TYPE "UDT_VfdNordParameter"
TITLE = UDT_VfdNordParameter
VERSION : 0.1
//Parameter structure to read and write
   STRUCT
      WriteValue : DInt;   // Parameter value to write
      ActualValue : DInt;   // Actual value read from VFD
      ParaNumber : Int;   // Parameter number to access
      Index : Int;   // Parameter index number to access
      ParaSet : Int;   // Parameter set to acces
      Format32 { ExternalAccessible := 'False'; ExternalVisible := 'False'; ExternalWritable := 'False'} : Bool;   // 1 = Write the parameter in DWord format. 0 = Write the parameter in Word format
      WriteAccess { ExternalAccessible := 'False'; ExternalVisible := 'False'; ExternalWritable := 'False'} : Bool;   // 1 = Write the parameter. 0 = Read the parameter
      InUse { ExternalAccessible := 'False'; ExternalVisible := 'False'; ExternalWritable := 'False'} : Bool;   // 1 = Parameter is to be processed
      RamOnly { ExternalAccessible := 'False'; ExternalVisible := 'False'; ExternalWritable := 'False'} : Bool;   // 1 = Save parameter in RAM, 0 = Save parameter in RAM and EEPROM
   END_STRUCT;

END_TYPE

FUNCTION_BLOCK "FB_VfdNORDParaAcycWrite"
{ S7_Optimized_Access := 'FALSE' }
VERSION : 0.1
// ATTRIBUTES
// AUTO_NUMBER = True
// BLOCK_NUMBER = 35
// END_ATTRIBUTES
   VAR_INPUT
      HW_Identifier { ExternalAccessible := 'False'; ExternalVisible := 'False'; ExternalWritable := 'False'} : HW_IO;
      idi_Value { ExternalAccessible := 'False'; ExternalVisible := 'False'; ExternalWritable := 'False'} : DInt;
      ii_FISystembus { ExternalAccessible := 'False'; ExternalVisible := 'False'; ExternalWritable := 'False'} : Int := 1;
      ii_ParameterNumber { ExternalAccessible := 'False'; ExternalVisible := 'False'; ExternalWritable := 'False'} : Int;
      ii_ParameterIndex { ExternalAccessible := 'False'; ExternalVisible := 'False'; ExternalWritable := 'False'} : Int;
      ii_ParameterSet { ExternalAccessible := 'False'; ExternalVisible := 'False'; ExternalWritable := 'False'} : Int;
      ix_Execute { ExternalAccessible := 'False'; ExternalVisible := 'False'; ExternalWritable := 'False'} : Bool;
      ix_Parameter32Bit { ExternalAccessible := 'False'; ExternalVisible := 'False'; ExternalWritable := 'False'} : Bool;
      ix_RAM_Only { ExternalAccessible := 'False'; ExternalVisible := 'False'; ExternalWritable := 'False'} : Bool;
   END_VAR

   VAR_OUTPUT
      qx_Done { ExternalAccessible := 'False'; ExternalVisible := 'False'; ExternalWritable := 'False'} : Bool;
      qx_Busy { ExternalAccessible := 'False'; ExternalVisible := 'False'; ExternalWritable := 'False'} : Bool;
      qx_Error { ExternalAccessible := 'False'; ExternalVisible := 'False'; ExternalWritable := 'False'} : Bool;
      qdi_ValueRead { ExternalAccessible := 'False'; ExternalVisible := 'False'; ExternalWritable := 'False'} : DInt;
      qw_ErrorID { ExternalAccessible := 'False'; ExternalVisible := 'False'; ExternalWritable := 'False'} : Word;
   END_VAR

   VAR
      sa_WriteVal { ExternalAccessible := 'False'; ExternalVisible := 'False'; ExternalWritable := 'False'} : Array[0..3] of Word;
      sa_RecWrite { ExternalAccessible := 'False'; ExternalVisible := 'False'; ExternalWritable := 'False'} AT sa_WriteVal : Struct
         PKE { ExternalAccessible := 'False'; ExternalVisible := 'False'; ExternalWritable := 'False'} : Word;
         Index { ExternalAccessible := 'False'; ExternalVisible := 'False'; ExternalWritable := 'False'} : Word;
         Para_Val { ExternalAccessible := 'False'; ExternalVisible := 'False'; ExternalWritable := 'False'} : DInt;
      END_STRUCT;
      sa_ReadVal { ExternalAccessible := 'False'; ExternalVisible := 'False'; ExternalWritable := 'False'} : Array[0..3] of Word;
      sa_RecRead { ExternalAccessible := 'False'; ExternalVisible := 'False'; ExternalWritable := 'False'} AT sa_ReadVal : Struct
         PKE { ExternalAccessible := 'False'; ExternalVisible := 'False'; ExternalWritable := 'False'} : Word;
         Index { ExternalAccessible := 'False'; ExternalVisible := 'False'; ExternalWritable := 'False'} : Word;
         Para_Val { ExternalAccessible := 'False'; ExternalVisible := 'False'; ExternalWritable := 'False'} : DInt;
      END_STRUCT;
      sv_WRRECInstance {InstructionName := 'WRREC'; LibVersion := '1.1'; ExternalAccessible := 'False'; ExternalVisible := 'False'; ExternalWritable := 'False'; S7_SetPoint := 'False'} : WRREC;
      sv_RDRECInstance {InstructionName := 'RDREC'; LibVersion := '1.0'; ExternalAccessible := 'False'; ExternalVisible := 'False'; ExternalWritable := 'False'; S7_SetPoint := 'False'} : RDREC;
      sw_Ak { ExternalAccessible := 'False'; ExternalVisible := 'False'; ExternalWritable := 'False'} : Word;
      sw_Pnu { ExternalAccessible := 'False'; ExternalVisible := 'False'; ExternalWritable := 'False'} : Word;
      sw_ErrorIDStatic { ExternalAccessible := 'False'; ExternalVisible := 'False'; ExternalWritable := 'False'} : Word;
      sdi_DataRecord { ExternalAccessible := 'False'; ExternalVisible := 'False'; ExternalWritable := 'False'} : DInt;
      si_Receivecounter { ExternalAccessible := 'False'; ExternalVisible := 'False'; ExternalWritable := 'False'} : Int;
      si_State { ExternalAccessible := 'False'; ExternalVisible := 'False'; ExternalWritable := 'False'} : Int;
      sx_FLMExecute { ExternalAccessible := 'False'; ExternalVisible := 'False'; ExternalWritable := 'False'} : Bool;
      sx_REdgeExecute { ExternalAccessible := 'False'; ExternalVisible := 'False'; ExternalWritable := 'False'} : Bool;
      sx_DoneStatic { ExternalAccessible := 'False'; ExternalVisible := 'False'; ExternalWritable := 'False'} : Bool;
      sx_ErrorStatic { ExternalAccessible := 'False'; ExternalVisible := 'False'; ExternalWritable := 'False'} : Bool;
   END_VAR

   VAR_TEMP
      tw_ResponseIND : Word;
      tw_ResponseLABEL : Word;
      tw_ResponsePNU : Word;
      tdi_ResponsePWE : DInt;
      tx_WithIndex : Bool;
      tx_WithParameterSet : Bool;
   END_VAR

   VAR CONSTANT
      cw_ChangeParameterValueWordEEPROM : Word := 2;
      cw_ChangeParameterValueWordRAM : Word := 14;
      cw_ChangeParameterValueDoubleWordEEPROM : Word := 3;
      cw_ChangeParameterValueDoubleWordRAM : Word := 13;
      cw_IncorretSubindex : Word := 3;
      cw_InternalResponseLabelCannotBeDepicted : Word := 202;
      cw_InvalidDataType : Word := 5;
      cw_NoResponse : Word := 0;
      cw_OrderCannotBeExecuted : Word := 7;
      cw_ParameterOffset : Word := 1000;
      cw_PNUMask : Word := 16#07FF;
      ci_ReceivecounterMax : Int := 255;
      ci_Length : UInt := 8;
   END_VAR


BEGIN
	(*
	----------------------------------------------------------------------------------------

	Version history:
	Date        | Version   | Author        | Remark
	----------------------------------------------------------------------------------------
	25/01/2021  | 0.1       | S.Theocharis  | Copy fron NORD library
	21/02/2023  | 4.0       | F.Baten       | 4.0 Release TIA 17.5
	*)
	// protects the frequency inverter from too frequent write requests.
	IF #ix_Execute <> #sx_FLMExecute THEN
	    IF #ix_Execute THEN
	        #sx_REdgeExecute := TRUE;
	    ELSE
	        #sx_REdgeExecute := FALSE;
	    END_IF;
	    #sx_FLMExecute := #ix_Execute;
	ELSE
	    #sx_REdgeExecute := FALSE;
	END_IF;

	#tx_WithIndex := #ii_ParameterIndex > 0;
	#tx_WithParameterSet := #ii_ParameterSet > 0;

	CASE #si_State OF

	    0:
	        IF #sx_REdgeExecute AND
	            NOT ((#ii_ParameterSet < 0) OR (#ii_ParameterIndex < 0) OR (#ii_ParameterSet > 4) OR
	            (#tx_WithParameterSet AND (#ii_ParameterIndex > 64)) OR (NOT #tx_WithParameterSet AND (#ii_ParameterIndex > 256)) OR
	            (NOT #ix_Parameter32Bit AND #idi_Value < -32768) OR (NOT #ix_Parameter32Bit AND #idi_Value > 16#FFFF)) THEN
	            //initialize
	            #sx_DoneStatic := FALSE;
	            #sx_ErrorStatic := FALSE;
	            #sw_ErrorIDStatic := 0;
	            #si_Receivecounter := 0;
	            #qx_Done := FALSE;
	            #qx_Busy := TRUE;

	            // get PROFINET IO data record
	            IF (#ii_ParameterNumber >= 150 AND #ii_ParameterNumber <= 199) OR (#ii_ParameterNumber >= 800 AND #ii_ParameterNumber <= 849) THEN
	                // order to the bus interface
	                #sdi_DataRecord := 100;
	            ELSIF ((#ii_ParameterNumber >= 0 AND #ii_ParameterNumber < 150) OR (#ii_ParameterNumber >= 200 AND #ii_ParameterNumber <= 799) OR
	                (#ii_ParameterNumber >= 850 AND #ii_ParameterNumber <= 999)) AND (#ii_FISystembus > 0) AND (#ii_FISystembus <= 8) THEN
	                // order to frequency inverter 1..8
	                #sdi_DataRecord := #ii_FISystembus + 100;
	            ELSE
	                #sdi_DataRecord := 0;
	            END_IF;

	            // get order label (AK)
	            IF #ix_RAM_Only THEN
	                IF #ix_Parameter32Bit THEN
	                    #sw_Ak := #cw_ChangeParameterValueDoubleWordRAM;
	                ELSE
	                    #sw_Ak := #cw_ChangeParameterValueWordRAM;
	                END_IF;
	            ELSE
	                IF #ix_Parameter32Bit THEN
	                    #sw_Ak := #cw_ChangeParameterValueDoubleWordEEPROM;
	                ELSE
	                    #sw_Ak := #cw_ChangeParameterValueWordEEPROM;
	                END_IF;
	            END_IF;

	            // merge parameter label (PKE)
	            #sw_Pnu := INT_TO_WORD(#ii_ParameterNumber + WORD_TO_INT(#cw_ParameterOffset));
	            #sa_RecWrite.PKE := SHL(IN := #sw_Ak, N := 12) OR #sw_Pnu;

	            // get sub-index (IND)
	            IF #tx_WithIndex AND #tx_WithParameterSet THEN
	                #sa_RecWrite.Index := SHL(IN := SHL(IN := INT_TO_WORD((#ii_ParameterIndex) - 1), N := 2) OR
	                                          INT_TO_WORD((#ii_ParameterSet) - 1), N := 8);
	            ELSIF NOT #tx_WithIndex AND #tx_WithParameterSet THEN
	                #sa_RecWrite.Index := SHL(IN := INT_TO_WORD((#ii_ParameterSet) - 1), N := 8);
	            ELSIF #tx_WithIndex AND NOT #tx_WithParameterSet THEN
	                #sa_RecWrite.Index := SHL(IN := INT_TO_WORD((#ii_ParameterIndex) - 1), N := 8);
	            ELSE
	                #sa_RecWrite.Index := 0;
	            END_IF;

	            // get parameter value (PWE)
	            #sa_RecWrite.Para_Val := #idi_Value;

	            // write data to device
	            #sv_WRRECInstance(REQ := TRUE,
	                              ID := #HW_Identifier,
	                              INDEX := #sdi_DataRecord,
	                              LEN := #ci_Length,
	                              DONE => #sv_WRRECInstance.DONE,
	                              BUSY => #sv_WRRECInstance.BUSY,
	                              ERROR => #sv_WRRECInstance.ERROR,
	                              RECORD := #sa_WriteVal);
	            #si_State := 1;
	        ELSIF #sx_REdgeExecute AND
	            ((#ii_ParameterSet < 0) OR (#ii_ParameterIndex < 0) OR (#ii_ParameterSet > 4) OR
	            (#tx_WithParameterSet AND (#ii_ParameterIndex > 63)) OR (NOT #tx_WithParameterSet AND (#ii_ParameterIndex > 255))) THEN
	            #sx_DoneStatic := FALSE;
	            #sx_ErrorStatic := TRUE;
	            #sw_ErrorIDStatic := #cw_IncorretSubindex;
	        ELSIF #sx_REdgeExecute AND
	            ((NOT #ix_Parameter32Bit AND #idi_Value < -32768) OR (NOT #ix_Parameter32Bit AND #idi_Value > 16#FFFF)) THEN
	            // limitation to int value range. positive hex crc checksums are allowed
	            #sx_DoneStatic := FALSE;
	            #sx_ErrorStatic := TRUE;
	            #sw_ErrorIDStatic := #cw_InvalidDataType;
	        ELSE
	            #sv_RDRECInstance(REQ := FALSE,
	                              ID := #HW_Identifier,
	                              INDEX := #sdi_DataRecord,
	                              MLEN := #ci_Length,
	                              RECORD := #sa_ReadVal);
	        END_IF;

	    1:
	        #sv_WRRECInstance();

	        IF #sv_WRRECInstance.DONE THEN
	            #sv_WRRECInstance(REQ := FALSE);
	            #si_State := 2;
	        ELSIF #sv_WRRECInstance.ERROR THEN
	            #sx_DoneStatic := FALSE;
	            #sx_ErrorStatic := TRUE;
	            #sw_ErrorIDStatic := DWORD_TO_WORD(#sv_WRRECInstance.STATUS);
	            #si_State := 0;
	            #qx_Done := FALSE;
	            #qx_Busy := TRUE;
	        END_IF;

	    2:
	        #sv_RDRECInstance(REQ := TRUE,
	                          ID := #HW_Identifier,
	                          INDEX := #sdi_DataRecord,
	                          MLEN := #ci_Length,
	                          RECORD := #sa_ReadVal);

	        #tw_ResponseLABEL := SHR(IN := #sa_RecRead.PKE, N := 12);
	        #tw_ResponsePNU := #sa_RecRead.PKE AND #cw_PNUMask;
	        #tw_ResponseIND := #sa_RecRead.Index;
	        #tdi_ResponsePWE := #sa_RecRead.Para_Val;
	        #qdi_ValueRead := #sa_RecRead.Para_Val;
	        IF #sv_RDRECInstance.ERROR THEN
	            #sx_DoneStatic := FALSE;
	            #sx_ErrorStatic := TRUE;
	            #sw_ErrorIDStatic := DWORD_TO_WORD(#sv_RDRECInstance.STATUS);
	            #si_State := 0;
	        ELSIF #sv_RDRECInstance.VALID AND #tw_ResponseLABEL = #cw_OrderCannotBeExecuted THEN
	            #sx_DoneStatic := FALSE;
	            #sx_ErrorStatic := TRUE;
	            #sw_ErrorIDStatic := DINT_TO_WORD(#tdi_ResponsePWE);
	            #si_State := 0;
	        ELSIF #sv_RDRECInstance.VALID AND #tw_ResponseLABEL <> #cw_NoResponse AND
	            #tw_ResponseLABEL <> #cw_OrderCannotBeExecuted AND #tw_ResponsePNU = #sw_Pnu AND
	            #tw_ResponseIND = #sa_RecWrite.Index THEN
	            // acyclic write command complete
	            #sx_DoneStatic := TRUE;
	            #si_State := 0;
	        END_IF;

	        // check for read timeout
	        IF #si_Receivecounter >= #ci_ReceivecounterMax THEN
	            #sx_DoneStatic := FALSE;
	            #sx_ErrorStatic := TRUE;
	            #sw_ErrorIDStatic := #cw_InternalResponseLabelCannotBeDepicted;
	            #si_State := 0;
	        ELSE
	            #si_Receivecounter := #si_Receivecounter + 1;
	        END_IF;
	END_CASE;

	// output assignment
	#qx_Busy := INT_TO_BOOL(#si_State) AND NOT #sx_DoneStatic AND NOT #sx_ErrorStatic;
	IF #ix_Execute THEN
	    #qx_Done := #sx_DoneStatic;
	    #qx_Error := #sx_ErrorStatic;
	    #qw_ErrorID := #sw_ErrorIDStatic;
	ELSE
	    #qx_Done := FALSE;
	    #qx_Error := FALSE;
	    #qw_ErrorID := 0;
	END_IF;
END_FUNCTION_BLOCK

TYPE "UDT_ConveyorStatus"
TITLE = UDT_ConveyorStatus
VERSION : 0.1
//User-defined structure of FB_Conveyor function block status.
   STRUCT
      Status : Int;   // Status number
      Specific : Struct
         Reverse { ExternalAccessible := 'False'; ExternalVisible := 'False'; ExternalWritable := 'False'} : Bool;   // Conveyor is running in reverse direction
      END_STRUCT;
   END_STRUCT;

END_TYPE

TYPE "UDT_PECStatus"
VERSION : 0.1
   STRUCT
      PEC { ExternalAccessible := 'False'; ExternalVisible := 'False'; ExternalWritable := 'False'} : Bool;   // Current state of the photo eye
      Jam { ExternalAccessible := 'False'; ExternalVisible := 'False'; ExternalWritable := 'False'} : Bool;   // PEC jam error
   END_STRUCT;

END_TYPE

FUNCTION_BLOCK "FB_VfdNORDParaAcycRead"
{ S7_Optimized_Access := 'FALSE' }
VERSION : 0.1
// ATTRIBUTES
// AUTO_NUMBER = True
// BLOCK_NUMBER = 34
// END_ATTRIBUTES
   VAR_INPUT
      iHW_Identifier { ExternalAccessible := 'False'; ExternalVisible := 'False'; ExternalWritable := 'False'} : HW_IO;
      ii_FISystembus { ExternalAccessible := 'False'; ExternalVisible := 'False'; ExternalWritable := 'False'} : Int := 1;
      ii_Parameter_Number { ExternalAccessible := 'False'; ExternalVisible := 'False'; ExternalWritable := 'False'} : Int;
      ii_Parameter_Index { ExternalAccessible := 'False'; ExternalVisible := 'False'; ExternalWritable := 'False'} : Int;
      ii_Parameter_Set { ExternalAccessible := 'False'; ExternalVisible := 'False'; ExternalWritable := 'False'} : Int;
      ix_Enable { ExternalAccessible := 'False'; ExternalVisible := 'False'; ExternalWritable := 'False'} : Bool;
   END_VAR

   VAR_OUTPUT
      qdi_Value { ExternalAccessible := 'False'; ExternalVisible := 'False'; ExternalWritable := 'False'} : DInt;
      qw_Error_ID { ExternalAccessible := 'False'; ExternalVisible := 'False'; ExternalWritable := 'False'} : Word;
      qx_Valid { ExternalAccessible := 'False'; ExternalVisible := 'False'; ExternalWritable := 'False'} : Bool;
      qx_Busy { ExternalAccessible := 'False'; ExternalVisible := 'False'; ExternalWritable := 'False'} : Bool;
      qx_Error { ExternalAccessible := 'False'; ExternalVisible := 'False'; ExternalWritable := 'False'} : Bool;
   END_VAR

   VAR
      sa_Write_Val { ExternalAccessible := 'False'; ExternalVisible := 'False'; ExternalWritable := 'False'} : Array[0..3] of Word;
      sa_Rec_Write { ExternalAccessible := 'False'; ExternalVisible := 'False'; ExternalWritable := 'False'} AT sa_Write_Val : Struct
         PKE { ExternalAccessible := 'False'; ExternalVisible := 'False'; ExternalWritable := 'False'} : Word;
         Index { ExternalAccessible := 'False'; ExternalVisible := 'False'; ExternalWritable := 'False'} : Word;
         Para_Val { ExternalAccessible := 'False'; ExternalVisible := 'False'; ExternalWritable := 'False'} : DInt;
      END_STRUCT;
      sa_Read_Val { ExternalAccessible := 'False'; ExternalVisible := 'False'; ExternalWritable := 'False'} : Array[0..3] of Word;
      sa_Rec_Read { ExternalAccessible := 'False'; ExternalVisible := 'False'; ExternalWritable := 'False'} AT sa_Read_Val : Struct
         PKE { ExternalAccessible := 'False'; ExternalVisible := 'False'; ExternalWritable := 'False'} : Word;
         Index { ExternalAccessible := 'False'; ExternalVisible := 'False'; ExternalWritable := 'False'} : Word;
         Para_Val { ExternalAccessible := 'False'; ExternalVisible := 'False'; ExternalWritable := 'False'} : DInt;
      END_STRUCT;
      sv_WRREC_Instance {InstructionName := 'WRREC'; LibVersion := '1.1'; ExternalAccessible := 'False'; ExternalVisible := 'False'; ExternalWritable := 'False'; S7_SetPoint := 'False'} : WRREC;
      sv_RDREC_Instance {InstructionName := 'RDREC'; LibVersion := '1.0'; ExternalAccessible := 'False'; ExternalVisible := 'False'; ExternalWritable := 'False'; S7_SetPoint := 'False'} : RDREC;
      sw_Ak { ExternalAccessible := 'False'; ExternalVisible := 'False'; ExternalWritable := 'False'} : Word;
      sdi_Data_Record { ExternalAccessible := 'False'; ExternalVisible := 'False'; ExternalWritable := 'False'} : DInt;
      sdi_ValueStatic { ExternalAccessible := 'False'; ExternalVisible := 'False'; ExternalWritable := 'False'} : DInt;
      sw_Pnu { ExternalAccessible := 'False'; ExternalVisible := 'False'; ExternalWritable := 'False'} : Word;
      sw_ErrorIDStatic { ExternalAccessible := 'False'; ExternalVisible := 'False'; ExternalWritable := 'False'} : Word;
      si_Receivecounter { ExternalAccessible := 'False'; ExternalVisible := 'False'; ExternalWritable := 'False'} : Int;
      si_State { ExternalAccessible := 'False'; ExternalVisible := 'False'; ExternalWritable := 'False'} : Int;
      sx_ValidStatic { ExternalAccessible := 'False'; ExternalVisible := 'False'; ExternalWritable := 'False'} : Bool;
      sx_ErrorStatic { ExternalAccessible := 'False'; ExternalVisible := 'False'; ExternalWritable := 'False'} : Bool;
   END_VAR

   VAR_TEMP
      tw_ResponseIND : Word;
      tw_ResponseLABEL : Word;
      tw_ResponsePNU : Word;
      tdi_ResponsePWE : DInt;
      tx_WithIndex : Bool;
      tx_WithParameterSet : Bool;
   END_VAR

   VAR CONSTANT
      cw_IncorrectSubindex : Word := 3;
      cw_InternalResponseLabelCannotBeDepicted : Word := 202;
      cw_NoResponse : Word := 0;
      cw_OrderCannotBeExecuted : Word := 7;
      cw_OrderParameterValue : Word := 1;
      cw_ParameterOffset : Word := 1000;
      cw_PNUMask : Word := 16#07FF;
      ci_ReceivecounterMax : Int := 255;
      ci_Length : UInt := 8;
   END_VAR


BEGIN
	(*
	----------------------------------------------------------------------------------------

	Version history:
	Date        | Version   | Author        | Remark
	----------------------------------------------------------------------------------------
	25/01/2021  | 0.1       | S.Theocharis  | Copy from NORD library
	21/02/2023  | 4.0       | F.Baten       | 4.0 Release TIA 17.5
	*)

	#tx_WithIndex := #ii_Parameter_Index > 0;
	#tx_WithParameterSet := #ii_Parameter_Set > 0;

	CASE #si_State OF

	    0:
	        IF #ix_Enable AND
	            NOT ((#ii_Parameter_Set < 0) OR (#ii_Parameter_Index < 0) OR (#ii_Parameter_Set > 4) OR
	            (#tx_WithParameterSet AND (#ii_Parameter_Index > 64)) OR (NOT #tx_WithParameterSet AND (#ii_Parameter_Index > 256))) THEN
	            //initialize
	            #si_Receivecounter := 0;

	            // get PROFINET IO data record
	            IF (#ii_Parameter_Number >= 150 AND #ii_Parameter_Number <= 199) OR (#ii_Parameter_Number >= 800 AND #ii_Parameter_Number <= 849) THEN
	                // order to the bus interface
	                #sdi_Data_Record := 100;
	            ELSIF ((#ii_Parameter_Number >= 0 AND #ii_Parameter_Number < 150) OR (#ii_Parameter_Number >= 200 AND #ii_Parameter_Number <= 799) OR
	                (#ii_Parameter_Number >= 850 AND #ii_Parameter_Number <= 999)) AND (#ii_FISystembus > 0) AND (#ii_FISystembus <= 8) THEN
	                // order to frequency inverter 1..8
	                #sdi_Data_Record := #ii_FISystembus + 100;
	            ELSE
	                #sdi_Data_Record := 0;
	            END_IF;

	            // get order label (AK)
	            #sw_Ak := #cw_OrderParameterValue;

	            // merge parameter label (PKE)
	            #sw_Pnu := INT_TO_WORD(#ii_Parameter_Number + WORD_TO_INT(#cw_ParameterOffset));
	            #sa_Rec_Write.PKE := SHL(IN := #sw_Ak, N := 12) OR #sw_Pnu;

	            // get sub-index (IND)
	            IF #tx_WithIndex AND #tx_WithParameterSet THEN
	                #sa_Rec_Write.Index := SHL(IN := SHL(IN := INT_TO_WORD((#ii_Parameter_Index) - 1), N := 2) OR
	                                           INT_TO_WORD((#ii_Parameter_Set) - 1), N := 8);
	            ELSIF NOT #tx_WithIndex AND #tx_WithParameterSet THEN
	                #sa_Rec_Write.Index := SHL(IN := INT_TO_WORD((#ii_Parameter_Set) - 1), N := 8);
	            ELSIF #tx_WithIndex AND NOT #tx_WithParameterSet THEN
	                #sa_Rec_Write.Index := SHL(IN := INT_TO_WORD((#ii_Parameter_Index) - 1), N := 8);
	            ELSE
	                #sa_Rec_Write.Index := 0;
	            END_IF;

	            // check if parameter or index changed from last request
	            IF (#sa_Rec_Read.PKE AND #cw_PNUMask) <> (#sa_Rec_Write.PKE AND #cw_PNUMask) OR
	                (#sa_Rec_Read.Index <> #sa_Rec_Write.Index) THEN
	                // if changed reset valid bit
	                #sx_ValidStatic := FALSE;
	                #sx_ErrorStatic := FALSE;
	            END_IF;

	            // write data to device
	            #sv_WRREC_Instance(REQ := TRUE,
	                               ID := #iHW_Identifier,
	                               INDEX := #sdi_Data_Record,
	                               LEN := #ci_Length,
	                               DONE => #sv_WRREC_Instance.DONE,
	                               BUSY => #sv_WRREC_Instance.BUSY,
	                               ERROR => #sv_WRREC_Instance.ERROR,
	                               RECORD := #sa_Write_Val);
	            #si_State := 1;
	        ELSIF #ix_Enable AND
	            ((#ii_Parameter_Set < 0) OR (#ii_Parameter_Index < 0) OR (#ii_Parameter_Set > 4) OR
	            (#tx_WithParameterSet AND (#ii_Parameter_Index > 63)) OR (NOT #tx_WithParameterSet AND (#ii_Parameter_Index > 255))) THEN
	            #sx_ValidStatic := FALSE;
	            #sx_ErrorStatic := TRUE;
	            #sdi_ValueStatic := 0;
	            #sw_ErrorIDStatic := #cw_IncorrectSubindex;
	        ELSE
	            #sv_RDREC_Instance(REQ := FALSE,
	                               ID := #iHW_Identifier,
	                               INDEX := #sdi_Data_Record,
	                               MLEN := #ci_Length,
	                               RECORD := #sa_Read_Val);
	            #sx_ValidStatic := FALSE;
	            #sx_ErrorStatic := FALSE;
	            #sw_ErrorIDStatic := 0;
	            #sdi_ValueStatic := 0;
	        END_IF;

	    1:
	        #sv_WRREC_Instance();

	        IF #sv_WRREC_Instance.DONE THEN
	            #sv_WRREC_Instance(REQ := FALSE);
	            #si_State := 2;
	        ELSIF #sv_WRREC_Instance.ERROR THEN
	            #sx_ValidStatic := FALSE;
	            #sx_ErrorStatic := TRUE;
	            #sdi_ValueStatic := 0;
	            #sw_ErrorIDStatic := DWORD_TO_WORD(#sv_WRREC_Instance.STATUS);
	            #si_State := 0;
	        END_IF;

	    2:
	        #sv_RDREC_Instance(REQ := TRUE,
	                           ID := #iHW_Identifier,
	                           INDEX := #sdi_Data_Record,
	                           MLEN := #ci_Length,
	                           RECORD := #sa_Read_Val);

	        #tw_ResponseLABEL := SHR(IN := #sa_Rec_Read.PKE, N := 12);
	        #tw_ResponsePNU := #sa_Rec_Read.PKE AND #cw_PNUMask;
	        #tw_ResponseIND := #sa_Rec_Read.Index;
	        #tdi_ResponsePWE := #sa_Rec_Read.Para_Val;

	        IF #sv_RDREC_Instance.ERROR THEN
	            #sx_ValidStatic := FALSE;
	            #sx_ErrorStatic := TRUE;
	            #sdi_ValueStatic := 0;
	            #sw_ErrorIDStatic := DWORD_TO_WORD(#sv_RDREC_Instance.STATUS);
	            #si_State := 0;
	        ELSIF #sv_RDREC_Instance.VALID AND #tw_ResponseLABEL = #cw_OrderCannotBeExecuted THEN
	            #sx_ValidStatic := FALSE;
	            #sx_ErrorStatic := TRUE;
	            #sdi_ValueStatic := 0;
	            #sw_ErrorIDStatic := DINT_TO_WORD(#tdi_ResponsePWE);
	            #si_State := 0;
	        ELSIF #sv_RDREC_Instance.VALID AND #tw_ResponseLABEL <> #cw_NoResponse AND
	            #tw_ResponseLABEL <> #cw_OrderCannotBeExecuted AND #tw_ResponsePNU = #sw_Pnu AND
	            #tw_ResponseIND = #sa_Rec_Write.Index THEN
	            // acyclic read command complete
	            #sx_ValidStatic := TRUE;
	            #sx_ErrorStatic := FALSE;
	            #sdi_ValueStatic := #tdi_ResponsePWE;
	            #sw_ErrorIDStatic := 0;
	            #si_State := 0;
	        END_IF;

	        // check for read timeout
	        IF #si_Receivecounter >= #ci_ReceivecounterMax THEN
	            #sx_ValidStatic := FALSE;
	            #sx_ErrorStatic := TRUE;
	            #sdi_ValueStatic := 0;
	            #sw_ErrorIDStatic := #cw_InternalResponseLabelCannotBeDepicted;
	            #si_State := 0;
	        ELSE
	            #si_Receivecounter := #si_Receivecounter + 1;
	        END_IF;

	END_CASE;

	// output assignment
	#qx_Busy := INT_TO_BOOL(#si_State);
	IF #ix_Enable THEN
	    #qx_Valid := #sx_ValidStatic;
	    #qx_Error := #sx_ErrorStatic;
	    #qw_Error_ID := #sw_ErrorIDStatic;
	    #qdi_Value := #sdi_ValueStatic;
	ELSE
	    #qx_Valid := FALSE;
	    #qx_Error := FALSE;
	    #qw_Error_ID := 0;
	    #qdi_Value := 0;
	END_IF;
END_FUNCTION_BLOCK

TYPE "UDT_ConveyorCommand"
TITLE = UDT_ConveyorCommand
VERSION : 0.1
//User-defined structure of conveyor commands.
   STRUCT
      ManualMode { ExternalAccessible := 'False'; ExternalVisible := 'False'; ExternalWritable := 'False'} : Bool;   // Manual mode command from HMI
      ManualStartStop { ExternalAccessible := 'False'; ExternalVisible := 'False'; ExternalWritable := 'False'} : Bool;   // Run conveyor in manual mode
      ManualFullSpeed { ExternalAccessible := 'False'; ExternalVisible := 'False'; ExternalWritable := 'False'} : Bool;   // Full speed conveyor in manual mode
      ManualJog { ExternalAccessible := 'False'; ExternalVisible := 'False'; ExternalWritable := 'False'} : Bool;   // Command to jog conveyor in slow speed from HMI
      Reverse { ExternalAccessible := 'False'; ExternalVisible := 'False'; ExternalWritable := 'False'} : Bool;   // Command to run conveyor in reverse direction from HMI
      ManualSpeed : Int := 50;   // Manual mode speed as percentage of nominal speed [0-100%]
   END_STRUCT;

END_TYPE

TYPE "UDT_RATStatistics"
VERSION : 0.1
   STRUCT
      AirPressure { S7_SetPoint := 'False'} : "UDT_EventStatistic";
      DivertUpError : "UDT_EventStatistic";
      DivertDownError : "UDT_EventStatistic";
      ConveyorUp : "UDT_EventStatistic";
      ConveyorDown : "UDT_EventStatistic";
      ConveyorStop : "UDT_EventStatistic";
   END_STRUCT;

END_TYPE

TYPE "UDT_ConveyorHandshake"
TITLE = UDT_ConveyorHandshake
VERSION : 0.1
//User-defined structure of conveyor handshake variables.
   STRUCT
      GIN : Int;   // General identification number
      NrOfPosToShift : Int;   // Number of positions to shift
      DownstreamDisplacement : Int;   // Displacement from downstream [cm]
      RTS { ExternalAccessible := 'False'; ExternalVisible := 'False'; ExternalWritable := 'False'} : Bool;   // Conveyor ready to send
      RTR { ExternalAccessible := 'False'; ExternalVisible := 'False'; ExternalWritable := 'False'} : Bool;   // Conveyor ready to receive
      TIP { ExternalAccessible := 'False'; ExternalVisible := 'False'; ExternalWritable := 'False'} : Bool;   // Transfer in progress
      ResetEnergySave { ExternalAccessible := 'False'; ExternalVisible := 'False'; ExternalWritable := 'False'} : Bool;   // Reset energy save mode
      CascadeStartUp { ExternalAccessible := 'False'; ExternalVisible := 'False'; ExternalWritable := 'False'} : Bool;   // Cascade startup
      ReqStop { ExternalAccessible := 'False'; ExternalVisible := 'False'; ExternalWritable := 'False'} : Bool;   // Request stop
   END_STRUCT;

END_TYPE

TYPE "UDT_ConveyorStatistics"
TITLE = UDT_ConveyorStatistics
VERSION : 0.1
//User-defined structure of FB_Conveyor function block statistics.
   STRUCT
      EnergySave : "UDT_EventStatistic";   // Number of times that save energy mode occurs
      ConveyorUp : "UDT_EventStatistic";   // Conveyor up statistics
      ConveyorDown : "UDT_EventStatistic";   // Conveyor down statistics
      ConveyorStop : "UDT_EventStatistic";   // Conveyor down statistics
   END_STRUCT;

END_TYPE

TYPE "UDT_VfdStatistics"
TITLE = UDT_VFDStatistics_SEW
VERSION : 0.1
//User-defined structure of FB_VFD_SEW_MOVI-C function block statistics.
   STRUCT
      PNSlaveNotOnline : "UDT_EventStatistic";   // Statistics of Profinet slave not online
      PNSlaveError : "UDT_EventStatistic";   // Statistics of a Profinet slave error
      VFDInternalError : "UDT_EventStatistic";   // Statistics of an internal VFD error
      CommunicationErrorMovikit : "UDT_EventStatistic";   // Statistics of a communication error
      Running : "UDT_EventStatistic";   // Statistics for running time
   END_STRUCT;

END_TYPE

TYPE "UDT_MotorData"
VERSION : 0.1
   STRUCT
      MainVoltage : Int;   // [Volt] Mains
      NominalVoltage : Int;   // [Volt] Motor nameplate for applicable connection
      NominalCurrent : Real;   // [Amps] Motor nameplate for applicable connection
      NominalPower : Real;   // [kW] Motor nameplate
      NominalSpeed : Int;   // [RPM] Motor nameplate
      NominalTorque : Real;   // [Nm] Motor nameplate
      CosPhi : Real;   // 0.0 - 0.99 Motor nameplate
      Connection : Int;   // 0=Start , 1=Delta
      BrakeConfig { ExternalAccessible := 'False'; ExternalVisible := 'False'; ExternalWritable := 'False'} : Bool;   // TRUE = Brake control from VFD. FALSE = No Brake
      EncoderConfig { ExternalAccessible := 'False'; ExternalVisible := 'False'; ExternalWritable := 'False'} : Bool;   // TRUE = Encoder connected at the VFD . FALSE = No encoder at the VFD
      EncoderResolution : Int;   // Pulses Per Rev
      ThermalConfig : Int;   // 0=No thermal control, 1= PTC1, 2=KTY84, 4= Bimetalic Switch
      NoMotorsParallel : Int;   // Number of motors in parallel
      VFDType : Int;   // Specific code 1= G120C, 5302= G120D 0,75kW, 5304= G120D 1,5kW, 5306= G120D 3kW, 5307= G120D 4kW, 5308= 5,5kW, 5309= G120D 7,5kW
      MinimumRamp : Int;   // Minimum applicable ramp in ms
      FAdress : Real;   // Safety adress from HW configuration
   END_STRUCT;

END_TYPE

TYPE "UDT_StatusTC07"
VERSION : 0.1
//One direction, motor, controler, EOS
   STRUCT
      Conveyor { ExternalWritable := 'False'} : "UDT_ConveyorStatus";   // Conveyor Status
      PEC_EoS { ExternalWritable := 'False'} : "UDT_PECStatus";   // PEC EoS Status
      MCO_M01 { ExternalWritable := 'False'} : "UDT_AixControllerStatus";   // MCO Status
      BladeStopEoS { ExternalWritable := 'False'} : "UDT_ValveStatus";   // Stop blade at the end of section status
   END_STRUCT;

END_TYPE

FUNCTION "FC_ExtractCodeFromString" : Void
{ S7_Optimized_Access := 'TRUE' }
VERSION : 0.1
   VAR_INPUT
      is_String : String;
   END_VAR

   VAR_OUTPUT
      qs_String : String;
   END_VAR

   VAR_TEMP
      ts_String : Bool;
      ti_StartPoint : Int;
      ti_StopPoint : Int;
      ti_CodeLenght : Int;
   END_VAR

   VAR CONSTANT
      StartSign : String := '$02';
      StopSign : String := '$03';
   END_VAR


BEGIN
	#ti_StartPoint := FIND(IN1 := #is_String, IN2 := #StartSign);
	#ti_StopPoint := FIND(IN1 := #is_String, IN2 := #StopSign);
	#ti_CodeLenght := #ti_StopPoint - #ti_StartPoint - 1;

	#qs_String := MID(IN := #is_String, L := #ti_CodeLenght, P := #ti_StartPoint + 1);

END_FUNCTION

TYPE "UDT_DataLogic_IN"
VERSION : 0.1
   STRUCT
      DataFromCamera : Byte;   // OK_READ - .%X0; NO_READ -.%X1; PhaseON -.%X3; PhaseOFF .%X4
      BarCodeValue0 : Byte;   // First character of the barcode.
      BarCodeValue : Array[1..14] of Char;   // Remaining characters of the barcode, after the barcode remaining chars are  '$00' = BYTE#16#00
   END_STRUCT;

END_TYPE

TYPE "UDT_StatusTC02"
VERSION : 0.1
//One direction, motor, controler, EOS
   STRUCT
      Conveyor : "UDT_ConveyorStatus";   // Conveyor Status
      PEC_EoS : "UDT_PECStatus";   // PEC EoS Status
      MCO_M01 : "UDT_AixControllerStatus";   // MCO Status
   END_STRUCT;

END_TYPE

TYPE "UDT_StatusTC12"
VERSION : 0.1
//One direction, motor, controler, EOS
   STRUCT
      Conveyor : "UDT_ConveyorStatus";   // Conveyor Status
      PEC_EoS : "UDT_PECStatus";   // PEC EoS Status
      MCO_M01 : "UDT_AixControllerStatus";   // MCO Status
   END_STRUCT;

END_TYPE

TYPE "UDT_StatusTC03"
VERSION : 0.1
//One direction, motor, controler, EOS, Tracking
//
   STRUCT
      Conveyor : "UDT_ConveyorStatus";   // Conveyor Status
      PEC_EoS : "UDT_PECUpdateStatus";   // PEC EoS Status
      MCO_M01 : "UDT_AixControllerStatus";   // MCO Status
   END_STRUCT;

END_TYPE

FUNCTION_BLOCK "SICK_Lector_CLV6xx_PNDP"
TITLE = SICK Lector6xx / CLV6xx function block
{ S7_Optimized_Access := 'TRUE' }
AUTHOR : SICKAG
FAMILY : Ident
VERSION : 1.2
// ATTRIBUTES
// AUTO_NUMBER = True
// BLOCK_NUMBER = 267
// END_ATTRIBUTES
//This function block is used for a communication between a SICK Lector6xx / SICK CLV6xx code reader and a Siemens S7-1200/S7-1500 PLC via  PROFINET/PROFIBUS
   VAR_INPUT
      HWInputIdent { ExternalAccessible := 'False'; ExternalVisible := 'False'; ExternalWritable := 'False'} : HW_IO;   // Hardware identification number of the input module
      HWInputLength { ExternalAccessible := 'False'; ExternalVisible := 'False'; ExternalWritable := 'False'} : USInt;   // Size of the input module
      HWOutputIdent { ExternalAccessible := 'False'; ExternalVisible := 'False'; ExternalWritable := 'False'} : HW_IO;   // Hardware identification number of the output module
      HWOutputLength { ExternalAccessible := 'False'; ExternalVisible := 'False'; ExternalWritable := 'False'} : USInt;   // Size of the output module
      CANId { ExternalAccessible := 'False'; ExternalVisible := 'False'; ExternalWritable := 'False'} : USInt;   // CAN ID (0= Master / No CAN network)
      TOut { ExternalAccessible := 'False'; ExternalVisible := 'False'; ExternalWritable := 'False'} : Time := T#10S;   // Time out
      Req { ExternalAccessible := 'False'; ExternalVisible := 'False'; ExternalWritable := 'False'} : Bool;   // A positive edge starts the request
      TriggerOn { ExternalAccessible := 'False'; ExternalVisible := 'False'; ExternalWritable := 'False'} : Bool;   // Select: Trigger On to open the reading gate via a SW-Trigger command
      TriggerOff { ExternalAccessible := 'False'; ExternalVisible := 'False'; ExternalWritable := 'False'} : Bool;   // Select: Trigger Off to close the reading gate via a SW-Trigger command
      Matchcode { ExternalAccessible := 'False'; ExternalVisible := 'False'; ExternalWritable := 'False'} : Bool;   // Select: Matchcode (details at #Data)
      SavePermanent { ExternalAccessible := 'False'; ExternalVisible := 'False'; ExternalWritable := 'False'} : Bool;   // Select: Save permanent
      ComTest { ExternalAccessible := 'False'; ExternalVisible := 'False'; ExternalWritable := 'False'} : Bool;   // Select: Communication test
      FreeCommand { ExternalAccessible := 'False'; ExternalVisible := 'False'; ExternalWritable := 'False'} : Bool;   // Select: Free command (details at #Data)
   END_VAR

   VAR_OUTPUT
      RdDone { ExternalAccessible := 'False'; ExternalVisible := 'False'; ExternalWritable := 'False'} : Bool;   // Positive edge: A reading result sent by the device was received
      ReqDone { ExternalAccessible := 'False'; ExternalVisible := 'False'; ExternalWritable := 'False'} : Bool;   // Request done
      ReqBusy { ExternalAccessible := 'False'; ExternalVisible := 'False'; ExternalWritable := 'False'} : Bool;   // Request in process
      Error { ExternalAccessible := 'False'; ExternalVisible := 'False'; ExternalWritable := 'False'} : Bool;   // Error detected
      Errorcode { ExternalAccessible := 'False'; ExternalVisible := 'False'; ExternalWritable := 'False'} : DWord;   // Error code (see documentation)
   END_VAR

   VAR_IN_OUT
      Data : "ST_SICK_Lector_CLV6xx";   // Command arguments and result outputs of the FB actions
   END_VAR

   VAR
      bTriggerReq { ExternalAccessible := 'False'; ExternalVisible := 'False'; ExternalWritable := 'False'} : Bool;   // Rising edge detection
      bTriggerReqMem { ExternalAccessible := 'False'; ExternalVisible := 'False'; ExternalWritable := 'False'} : Bool;   // Rising edge detection
      bTriggerDone { ExternalAccessible := 'False'; ExternalVisible := 'False'; ExternalWritable := 'False'} : Bool;   // Rising edge detection
      bTriggerDoneMem { ExternalAccessible := 'False'; ExternalVisible := 'False'; ExternalWritable := 'False'} : Bool;   // Rising edge detection
      bTriggerError { ExternalAccessible := 'False'; ExternalVisible := 'False'; ExternalWritable := 'False'} : Bool;   // Rising edge detection
      bTriggerErrorMem { ExternalAccessible := 'False'; ExternalVisible := 'False'; ExternalWritable := 'False'} : Bool;   // Rising edge detection
      bCanActive { ExternalAccessible := 'False'; ExternalVisible := 'False'; ExternalWritable := 'False'} : Bool;   // CAN-Bus active flag
      bDeviceState { ExternalAccessible := 'False'; ExternalVisible := 'False'; ExternalWritable := 'False'} : Bool;   // Current device state (True= Edit-Mode | False= Run-Mode)
      bEnforceLogout { ExternalAccessible := 'False'; ExternalVisible := 'False'; ExternalWritable := 'False'} : Bool;   // Logout enforced
      bReqBusyMem { ExternalAccessible := 'False'; ExternalVisible := 'False'; ExternalWritable := 'False'} : Bool;   // Backup variable
      iStep { ExternalAccessible := 'False'; ExternalVisible := 'False'; ExternalWritable := 'False'} : USInt;   // Currrent FB step
      iCommandIndex { ExternalAccessible := 'False'; ExternalVisible := 'False'; ExternalWritable := 'False'} : Int;   // Command index
      iCommandLength { ExternalAccessible := 'False'; ExternalVisible := 'False'; ExternalWritable := 'False'} : UInt;   // Length of the command that should be send
      iRecordSize { ExternalAccessible := 'False'; ExternalVisible := 'False'; ExternalWritable := 'False'} : UInt;   // Length of the record array
      iCommandSize { ExternalAccessible := 'False'; ExternalVisible := 'False'; ExternalWritable := 'False'} : UInt;   // Length of the command array
      iReadingResultSize { ExternalAccessible := 'False'; ExternalVisible := 'False'; ExternalWritable := 'False'} : UInt;   // Length of the reading result array
      iIndex { ExternalAccessible := 'False'; ExternalVisible := 'False'; ExternalWritable := 'False'} : UInt;   // Index variable
      nTempErrorCode { ExternalAccessible := 'False'; ExternalVisible := 'False'; ExternalWritable := 'False'} : DWord;   // Temporarily error code
      nLogoutErrorCode { ExternalAccessible := 'False'; ExternalVisible := 'False'; ExternalWritable := 'False'} : DWord;   // Temporarily error code
      arrSelection { ExternalAccessible := 'False'; ExternalVisible := 'False'; ExternalWritable := 'False'} : Array[0..5] of Bool;   // input bit selection
      arrCommand { ExternalAccessible := 'False'; ExternalVisible := 'False'; ExternalWritable := 'False'} : Array[0..499] of Byte;   // Contains the transmitted CoLa command
      arrRecord { ExternalAccessible := 'False'; ExternalVisible := 'False'; ExternalWritable := 'False'} : Array[0..499] of Byte;   // Contains the received telegram
      fbTimeout {InstructionName := 'TON_TIME'; LibVersion := '1.0'; ExternalAccessible := 'False'; ExternalVisible := 'False'; ExternalWritable := 'False'; S7_SetPoint := 'False'} : TON_TIME;   // Instance: Timer on delay (Time out)
      fbCCom { ExternalAccessible := 'False'; ExternalVisible := 'False'; ExternalWritable := 'False'; S7_SetPoint := 'False'} : "SICK_CCOMM_PNDP";   // Instance: CoLa communication block
   END_VAR

   VAR_TEMP
      iTemp1 : Int;   // Temporarily variable
      iTemp2 : UDInt;   // Temporarily variable
      iTemp3 : UDInt;   // Temporarily variable
      nFncValue : DWord;   // Get/Set function value
      nFncErrorCode : Word;   // Get/Set function error code
   END_VAR


BEGIN
	(*===========================================================================================
	Name:   SICK_Lector_CLV6xx_PNDP
	Author: SICK AG
	=============================================================================================
	Description:
	This function block is used for a communication between a SICK Lector6xx / SICK CLV6xx
	code reader and a Siemens S7-1200/S7-1500 PLC via PROFINET/PROFIBUS.

	=============================================================================================
	Features:
	- Receive reading results of the device, triggered by a command, fieldbus or by a hardware
	  switch. The content of the result can be modified in the "Output Format" option in the
	  SOPAS engineeringtool.
	- Open and close a reading gate (software trigger via command)
	- Set a new Matchcode evaluation condition
	- Save all device parameters permanent
	- Communication test
	- Send a free defined CoLa-A telegram and receive the result
	- All commands can also be used in a SICK CAN-Bus network

	=============================================================================================
	Version history:
	Date       | Version | Author  | Remark
	---------------------------------------------------------------------------------------------
	21/02/2014 | V1.0    | SICK AG | Initial version
	07/08/2014 | V1.1    | SICK AG | Replace R_TRIG function
	24/10/2017 | V1.2    | SICK AG | Avoid initialization warnings which occurs using TIA V13 or higher
	============================================================================================*)

	(*===================================== INITIALISATION =====================================*)
	#iRecordSize := 500;         (*Length of the arrRecord array*)
	#iCommandSize := 500;        (*Length of the arrCommand array*)
	#iReadingResultSize := 200;  (*Length of the reading result array*)

	(*Rising edge detection*)
	#bTriggerReq := #Req AND NOT #bTriggerReqMem;
	#bTriggerReqMem := #Req;
	#bTriggerDone := #fbCCom.ReqDone AND NOT #bTriggerDoneMem;
	#bTriggerDoneMem := #fbCCom.ReqDone;
	#bTriggerError := #fbCCom.Error AND NOT #bTriggerErrorMem;
	#bTriggerErrorMem := #fbCCom.Error;

	(*Reset the read done flag every cycle*)
	#RdDone := false;


	(*===================================== ERROR HANDLING =====================================*)
	(* bDeviceState  |  bEnforceLogout  |  Action
	       FALSE     |      FALSE       |  Errorcode = Errorcode from last plc cycle
	       FALSE     |      TRUE        |  Errorcode = Logout error
	       TRUE      |      FALSE       |  Enforce "Logout" command
	       TRUE      |      TRUE        |  Errorcode = Logout not possible + Reason*)
	IF #nTempErrorCode <> 16#0000_0000 THEN

	    (*Enfore "Logout" command*)
	    IF #bDeviceState AND NOT #bEnforceLogout THEN
	        #bEnforceLogout := true;
	        #iCommandIndex := 11;                  (*Logout*)
	        #nLogoutErrorCode := #nTempErrorCode;  (*Save current error code*)
	        #nTempErrorCode := 16#0000_0000;       (*Clear currenr error variable*)
	        #iStep := 4;                           (*Create command*)

	        (*Logout can not be ensured*)
	    ELSIF #bDeviceState AND #bEnforceLogout THEN
	        #Errorcode.%W1 := #nTempErrorCode.%W0;
	        #Errorcode.%W0 := 16#0017;  (*Error: Logout can not be ensured (please check the device state)*)

	        (*Errorcode = Errorcode from the last plc cycle or logout error*)
	    ELSE
	        #Errorcode := #nTempErrorCode;
	    END_IF;

	    (*Update FB status*)
	    IF #nTempErrorCode <> 16#0000_0000 THEN
	        #ReqDone := false;
	        #ReqBusy := false;
	        #bReqBusyMem := false;
	        #Error := true;
	        #nTempErrorCode := 16#0000_0000;
	        #nLogoutErrorCode := 16#0000_0000;
	        #iStep := 0;
	        RETURN;
	    END_IF;
	END_IF;

	(*Time out detection*)
	#fbTimeout(IN := #bReqBusyMem,
	           PT := #TOut);
	IF #fbTimeout.Q THEN
	    #nTempErrorCode := 16#0000_0010; (*Error: Time out*)
	END_IF;

	(*Check if a device error is detected: 'sFA XX'*)
	IF #bTriggerDone AND ((NOT #bCanActive AND
	    #arrRecord[0] = 's' AND
	    #arrRecord[1] = 'F' AND
	    #arrRecord[2] = 'A') OR (#bCanActive AND
	    #arrRecord[0] = 's' AND
	    #arrRecord[12] = 'F' AND
	    #arrRecord[13] = 'A')) THEN

	    (*Get the position of the error code*)
	    IF #bCanActive THEN
	        #iIndex := 15;
	    ELSE
	        #iIndex := 4;
	    END_IF;

	    "SICK_GetValue"(iTelegramLength := INT_TO_UINT(#fbCCom.ReqLength),
	                    iValueLength := 0,
	                    nValue => #nFncValue,
	                    nErrorCode => #nFncErrorCode,
	                    iPosition := #iIndex,
	                    arrData := #arrRecord);

	    IF #nFncErrorCode = 16#0000 THEN
	        #nTempErrorCode.%W1 := DWORD_TO_WORD(#nFncValue);
	        #nTempErrorCode.%W0 := 16#0011; (*Error: Device error*)
	    ELSE
	        #nTempErrorCode.%W1 := #nFncErrorCode;
	        #nTempErrorCode.%W0 := 16#0012; (*Error: SICK_GetValue error*)
	    END_IF;
	END_IF;

	(*Error detected*)
	IF #nTempErrorCode <> 16#0000_0000 THEN
	    RETURN;
	END_IF;


	(*================================= START REQUEST (STEP 1) =================================*)
	IF NOT #bReqBusyMem AND #bTriggerReq THEN
	    #ReqDone := false;
	    #ReqBusy := true;
	    #bReqBusyMem := true;
	    #Error := false;
	    #Errorcode := 16#0000_0000;
	    #bDeviceState := false;
	    #bEnforceLogout := false;

	    (*Save the current bit selection for the job*)
	    #arrSelection[0] := #TriggerOn;
	    #arrSelection[1] := #TriggerOff;
	    #arrSelection[2] := #Matchcode;
	    #arrSelection[3] := #SavePermanent;
	    #arrSelection[4] := #ComTest;
	    #arrSelection[5] := #FreeCommand;

	    (*Check CAN-ID*)
	    IF #CANId > 63 THEN
	        #nTempErrorCode := 16#0000_0014; (*Error invalid CAN Id*)
	    ELSIF #CANId = 0 THEN
	        #bCanActive := false;
	        #iStep := 3; (*Check parameter input*)
	    ELSE
	        #bCanActive := true;
	        #iStep := 2; (*Add CAN identifier*)
	    END_IF;
	END_IF;


	(*=============================== ADD CAN IDENTIFIER (STEP 2) ==============================*)
	IF #iStep = 2 THEN
	    Strg_TO_Chars(Strg := 's{ 00 01 ',
	                  pChars := 0,
	                  Cnt => #iIndex,
	                  Chars := #arrCommand);

	    "SICK_SetValue"(bAddBlank := false,
	                    nValue := #CANId,
	                    arrData => #arrCommand,
	                    nErrorCode => #nFncErrorCode,
	                    iPosition := #iIndex);
	    IF #nFncErrorCode <> 16#0000 THEN
	        #nTempErrorCode.%W1 := #nFncErrorCode;
	        #nTempErrorCode.%W0 := 16#0013; (*Error: SICK_SetValue error*)
	    ELSE
	        #arrCommand[#iIndex] := '}';
	        #iStep := 3; (*Check parameter input*)
	    END_IF;
	END_IF;


	(*============================= CHECK PARAMETER INPUT (STEP 3) =============================*)
	IF #iStep = 3 THEN
	    #iTemp1 := 0; (*Counts up the active bit selection*)

	    (*Command: Trigger On*)
	    IF #arrSelection[0] THEN
	        #iTemp1 := #iTemp1 + 1;
	        #iCommandIndex := 0; (*Send a "Trigger On" command*)
	    END_IF;

	    (*Command: Trigger Off*)
	    IF #arrSelection[1] THEN
	        #iTemp1 := #iTemp1 + 1;
	        #iCommandIndex := 1; (*Send a "Trigger Off" command*)
	    END_IF;

	    (*Command: Matchcode*)
	    IF #arrSelection[2] THEN
	        #iTemp1 := #iTemp1 + 1;

	        IF #Data.Matchcode.sName = '' THEN
	            #nTempErrorCode := 16#0000_0022; (*Error: Matchcode name is empty*)
	        ELSIF #Data.Matchcode.nCodeType <= '$20' OR #Data.Matchcode.nCodeType > '$7E' THEN
	            #nTempErrorCode := 16#0000_0023; (*Error: Invalid code type*)
	        END_IF;

	        #iCommandIndex := 10; (*Send a "Login" command*)
	    END_IF;

	    (*Command: Save permanent*)
	    IF #arrSelection[3] THEN
	        #iTemp1 := #iTemp1 + 1;
	        #iCommandIndex := 10; (*Send a "Login" command*)
	    END_IF;

	    (*Command: Communication test*)
	    IF #arrSelection[4] THEN
	        #iTemp1 := #iTemp1 + 1;
	        #iCommandIndex := 4; (*Send a "Comm Test" command*)
	    END_IF;

	    (*Command: Free command*)
	    IF #arrSelection[5] THEN
	        #iTemp1 := #iTemp1 + 1;

	        (*Check length*)
	        IF #bCanActive THEN
	            #iTemp2 := INT_TO_UDINT(LEN(#Data.FreeCommand.sCommand)) + 11;
	        ELSE
	            #iTemp2 := INT_TO_UDINT(LEN(#Data.FreeCommand.sCommand));
	        END_IF;

	        IF (LEN(#Data.FreeCommand.sCommand) <= 0) OR (#iTemp2 > #iCommandSize) THEN
	            #nTempErrorCode := 16#0000_0020; (*Error: Invalid free command length*)
	        END_IF;

	        #iCommandIndex := 5; (*Send a "Free Command" command*)
	    END_IF;

	    (*Check bit sum of the command selection*)
	    IF #iTemp1 <> 1 THEN
	        #nTempErrorCode := 16#0000_0015; (*Error: More than one or no parameter selected*)
	    END_IF;

	    (*Check if a error was detected*)
	    IF #nTempErrorCode = 16#0000_0000 THEN
	        #iStep := 4; (*Create CoLa command*)
	    END_IF;
	END_IF;


	(*============================== CREATE COLA COMMAND (STEP 4) ==============================*)
	IF #iStep = 4 THEN
	    CASE #iCommandIndex OF

	            (*Create "Trigger On" command*)
	        0:
	            IF #bCanActive THEN
	                Strg_TO_Chars(Strg := 'MN mTCgateon',
	                              pChars := 12,
	                              Cnt => #iTemp3,
	                              Chars := #arrCommand);
	                #iCommandLength := UDINT_TO_UINT(#iTemp3) + 12;
	            ELSE
	                Strg_TO_Chars(Strg := 'sMN mTCgateon',
	                              pChars := 0,
	                              Cnt => #iTemp3,
	                              Chars := #arrCommand);
	                #iCommandLength := UDINT_TO_UINT(#iTemp3);
	            END_IF;
	            #iStep := 5; (*Send command*)

	            (*Create "Trigger Off" command*)
	        1:
	            IF #bCanActive THEN
	                Strg_TO_Chars(Strg := 'MN mTCgateoff',
	                              pChars := 12,
	                              Cnt => #iTemp3,
	                              Chars := #arrCommand);
	                #iCommandLength := UDINT_TO_UINT(#iTemp3) + 12;
	            ELSE
	                Strg_TO_Chars(Strg := 'sMN mTCgateoff',
	                              pChars := 0,
	                              Cnt => #iTemp3,
	                              Chars := #arrCommand);
	                #iCommandLength := UDINT_TO_UINT(#iTemp3);
	            END_IF;
	            #iStep := 5; (*Send command*)

	            (*Create "Matchcode" command*)
	        2:
	            IF #bCanActive THEN
	                Strg_TO_Chars(Strg := 'MN mEVSetMatchCode 00 ',
	                              pChars := 12,
	                              Cnt => #iTemp3,
	                              Chars := #arrCommand);
	                #iIndex := UDINT_TO_UINT(#iTemp3 + 12);
	            ELSE
	                Strg_TO_Chars(Strg := 'sMN mEVSetMatchCode 00 ',
	                              pChars := 0,
	                              Cnt => #iTemp3,
	                              Chars := #arrCommand);
	                #iIndex := UDINT_TO_UINT(#iTemp3);
	            END_IF;

	            (*Add matchcode name*)
	            Strg_TO_Chars(Strg := CONCAT(IN1 := 'name="', IN2 := #Data.Matchcode.sName),
	                          pChars := #iIndex,
	                          Cnt => #iTemp3,
	                          Chars := #arrCommand);
	            #iIndex := #iIndex + UDINT_TO_UINT(#iTemp3);

	            (*Add codeType*)
	            Strg_TO_Chars(Strg := '" codeType="',
	                          pChars := #iIndex,
	                          Cnt => #iTemp3,
	                          Chars := #arrCommand);
	            #iIndex := #iIndex + UDINT_TO_UINT(#iTemp3);
	            IF #Data.Matchcode.nCodeType = '*' THEN
	                Strg_TO_Chars(Strg := 'dontCare',
	                              pChars := #iIndex,
	                              Cnt => #iTemp3,
	                              Chars := #arrCommand);
	                #iIndex := #iIndex + UDINT_TO_UINT(#iTemp3);
	            ELSE
	                #arrCommand[#iIndex] := #Data.Matchcode.nCodeType;
	                #iIndex := #iIndex + 1;
	            END_IF;

	            (*Add Min/Max length*)
	            Strg_TO_Chars(Strg := '" length="',
	                          pChars := #iIndex,
	                          Cnt => #iTemp3,
	                          Chars := #arrCommand);
	            #iIndex := #iIndex + UDINT_TO_UINT(#iTemp3);
	            IF #Data.Matchcode.iMinMaxLength = 0 THEN
	                Strg_TO_Chars(Strg := 'dontCare',
	                              pChars := #iIndex,
	                              Cnt => #iTemp3,
	                              Chars := #arrCommand);
	                #iIndex := #iIndex + UDINT_TO_UINT(#iTemp3);
	            ELSE
	                #arrCommand[#iIndex] := ((#Data.Matchcode.iMinMaxLength / 100) MOD 10) + 16#30;
	                #arrCommand[#iIndex + 1] := ((#Data.Matchcode.iMinMaxLength / 10) MOD 10) + 16#30;
	                #arrCommand[#iIndex + 2] := (#Data.Matchcode.iMinMaxLength MOD 10) + 16#30;
	                #iIndex := #iIndex + 3;
	            END_IF;

	            (*Add content*)
	            Strg_TO_Chars(Strg := CONCAT(IN1 := '" content="', IN2 := #Data.Matchcode.sContent),
	                          pChars := #iIndex,
	                          Cnt => #iTemp3,
	                          Chars := #arrCommand);
	            #iIndex := #iIndex + UDINT_TO_UINT(#iTemp3);
	            #arrCommand[#iIndex] := '"';


	            (*Overwrite the matchcode length*)
	            IF #bCanActive THEN
	                #nFncValue := #iIndex - 33;      (*Length of the #Matchcode command*)
	                #iCommandLength := #iIndex + 1;  (*Length of the whole CoLa command*)
	                #iIndex := 31;                 (*Startindex of the matchcode length*)
	            ELSE
	                #nFncValue := #iIndex - 22;      (*Length of the #Matchcode command*)
	                #iCommandLength := #iIndex + 1;  (*Length of the whole CoLa command*)
	                #iIndex := 20;                 (*Startindex of the matchcode length*)
	            END_IF;

	            "SICK_SetValue"(bAddBlank := false,
	                            nValue := #nFncValue,
	                            arrData => #arrCommand,
	                            nErrorCode => #nFncErrorCode,
	                            iPosition := #iIndex);
	            IF #nFncErrorCode <> 16#0000 THEN
	                #nTempErrorCode.%W1 := #nFncErrorCode;
	                #nTempErrorCode.%W0 := 16#0013; (*Error: SICK_SetValue error*)
	            ELSE
	                #iStep := 5; (*Send command*)
	            END_IF;

	            (*Create "Save Permanent" command*)
	        3:
	            IF #bCanActive THEN
	                Strg_TO_Chars(Strg := 'MN mEEwriteall',
	                              pChars := 12,
	                              Cnt => #iTemp3,
	                              Chars := #arrCommand);
	                #iCommandLength := UDINT_TO_UINT(#iTemp3 + 12);
	            ELSE
	                Strg_TO_Chars(Strg := 'sMN mEEwriteall',
	                              pChars := 0,
	                              Cnt => #iTemp3,
	                              Chars := #arrCommand);
	                #iCommandLength := UDINT_TO_UINT(#iTemp3);
	            END_IF;
	            #iStep := 5; (*Send command*)

	            (*Create "Communication Test" command*)
	        4:
	            IF #bCanActive THEN
	                Strg_TO_Chars(Strg := 'RI0',
	                              pChars := 12,
	                              Cnt => #iTemp3,
	                              Chars := #arrCommand);
	                #iCommandLength := UDINT_TO_UINT(#iTemp3) + 12;
	            ELSE
	                Strg_TO_Chars(Strg := 'sRI0',
	                              pChars := 0,
	                              Cnt => #iTemp3,
	                              Chars := #arrCommand);
	                #iCommandLength := UDINT_TO_UINT(#iTemp3);
	            END_IF;
	            #iStep := 5; (*Send command*)

	            (*Create "Free Command"*)
	        5:
	            IF #bCanActive THEN
	                Strg_TO_Chars(Strg := DELETE(IN := #Data.FreeCommand.sCommand, L := 1, P := 1),
	                              pChars := 12,
	                              Cnt => #iTemp3,
	                              Chars := #arrCommand);
	                #iCommandLength := UDINT_TO_UINT(#iTemp3) + 12;
	            ELSE
	                Strg_TO_Chars(Strg := #Data.FreeCommand.sCommand,
	                              pChars := 0,
	                              Cnt => #iTemp3,
	                              Chars := #arrCommand);
	                #iCommandLength := UDINT_TO_UINT(#iTemp3);
	            END_IF;
	            #iStep := 5; (*Send command*)

	            (*Create "Login" command*)
	        10:
	            IF #bCanActive THEN
	                Strg_TO_Chars(Strg := 'MN SetAccessMode 03 F4724744',
	                              pChars := 12,
	                              Cnt => #iTemp3,
	                              Chars := #arrCommand);
	                #iCommandLength := UDINT_TO_UINT(#iTemp3) + 12;
	            ELSE
	                Strg_TO_Chars(Strg := 'sMN SetAccessMode 03 F4724744',
	                              pChars := 0,
	                              Cnt => #iTemp3,
	                              Chars := #arrCommand);
	                #iCommandLength := UDINT_TO_UINT(#iTemp3);
	            END_IF;
	            #iStep := 5; (*Send command*)

	            (*Create "Logout" command*)
	        11:
	            IF #bCanActive THEN
	                Strg_TO_Chars(Strg := 'MN Run',
	                              pChars := 12,
	                              Cnt => #iTemp3,
	                              Chars := #arrCommand);
	                #iCommandLength := UDINT_TO_UINT(#iTemp3) + 12;
	            ELSE
	                Strg_TO_Chars(Strg := 'sMN Run',
	                              pChars := 0,
	                              Cnt => #iTemp3,
	                              Chars := #arrCommand);
	                #iCommandLength := UDINT_TO_UINT(#iTemp3);
	            END_IF;
	            #iStep := 5; (*Send command*)

	    END_CASE;
	END_IF;


	(*=============================== SEND COLA COMMAND (STEP 5) ===============================*)
	IF #iStep = 5 THEN
	    IF NOT #fbCCom.ReqBusy AND NOT #bTriggerDone AND NOT #bTriggerError THEN
	        #fbCCom.Req := true;
	        #iStep := 6; (*Wait for the command answer*)
	    END_IF;
	END_IF;


	(*========================== WAIT FOR THE COMMAND ANSWER (STEP 6) ==========================*)
	IF #iStep = 6 THEN
	    (*Communication error*)
	    IF #bTriggerError THEN
	        #nTempErrorCode := #fbCCom.Errorcode; (*Error: Communication error*)

	        (*Communication done*)
	    ELSIF #bTriggerDone THEN
	        #iStep := 7; (*Check the command answer*)
	    END_IF;
	END_IF;


	(*============================= CHECK COMMAND RESPONSE (STEP 7) ============================*)
	IF #iStep = 7 THEN
	    CASE #iCommandIndex OF

	            (*Check "Trigger On" response*)
	        0:
	            IF #bCanActive THEN
	                IF #arrRecord[0] = 's' AND
	                    #arrRecord[12] = 'A' AND
	                    #arrRecord[13] = 'N' AND
	                    #arrRecord[22] = 'o' AND
	                    #arrRecord[23] = 'n' AND
	                    #arrRecord[24] = ' ' AND
	                    #arrRecord[25] = '1' THEN

	                    #iStep := 8; (*Action performed*)
	                ELSE
	                    #nTempErrorCode := 16#0000_0016; (*Error: Invalid device answer*)
	                END_IF;
	            ELSE
	                IF #arrRecord[0] = 's' AND
	                    #arrRecord[1] = 'A' AND
	                    #arrRecord[2] = 'N' AND
	                    #arrRecord[11] = 'o' AND
	                    #arrRecord[12] = 'n' AND
	                    #arrRecord[13] = ' ' AND
	                    #arrRecord[14] = '1' THEN

	                    #iStep := 8; (*Action performed*)
	                ELSE
	                    #nTempErrorCode := 16#0000_0016; (*Error: Invalid device answer*)
	                END_IF;
	            END_IF;

	            (*Check "Trigger Off" response*)
	        1:
	            IF #bCanActive THEN
	                IF #arrRecord[0] = 's' AND
	                    #arrRecord[12] = 'A' AND
	                    #arrRecord[13] = 'N' AND
	                    #arrRecord[22] = 'o' AND
	                    #arrRecord[23] = 'f' AND
	                    #arrRecord[24] = 'f' AND
	                    #arrRecord[25] = ' ' AND
	                    #arrRecord[26] = '1' THEN

	                    #iStep := 8; (*Action performed*)
	                ELSE
	                    #nTempErrorCode := 16#0000_0016; (*Error: Invalid device answer*)
	                END_IF;
	            ELSE
	                IF #arrRecord[0] = 's' AND
	                    #arrRecord[1] = 'A' AND
	                    #arrRecord[2] = 'N' AND
	                    #arrRecord[11] = 'o' AND
	                    #arrRecord[12] = 'f' AND
	                    #arrRecord[13] = 'f' AND
	                    #arrRecord[14] = ' ' AND
	                    #arrRecord[15] = '1' THEN

	                    #iStep := 8; (*Action performed*)
	                ELSE
	                    #nTempErrorCode := 16#0000_0016; (*Error: Invalid device answer*)
	                END_IF;
	            END_IF;

	            (*Check "Matchcode" response*)
	        2:
	            IF #bCanActive THEN
	                IF NOT (#arrRecord[0] = 's' AND
	                    #arrRecord[12] = 'A' AND
	                    #arrRecord[13] = 'N' AND
	                    #arrRecord[27] = 'o' AND
	                    #arrRecord[28] = 'd' AND
	                    #arrRecord[29] = 'e' AND
	                    #arrRecord[30] = ' ' AND
	                    #arrRecord[31] = '1') THEN

	                    #nTempErrorCode := 16#0000_0016; (*Error: Invalid device answer*)
	                END_IF;
	            ELSE
	                IF NOT (#arrRecord[0] = 's' AND
	                    #arrRecord[1] = 'A' AND
	                    #arrRecord[2] = 'N' AND
	                    #arrRecord[16] = 'o' AND
	                    #arrRecord[17] = 'd' AND
	                    #arrRecord[18] = 'e' AND
	                    #arrRecord[19] = ' ' AND
	                    #arrRecord[20] = '1') THEN

	                    #nTempErrorCode := 16#0000_0016; (*Error: Invalid device answer*)
	                END_IF;
	            END_IF;

	            IF #nTempErrorCode = 0 THEN
	                #iCommandIndex := 11; (*Logout*)
	                #iStep := 4;         (*Create command*)
	            END_IF;

	            (*Check "Save Permanent" response*)
	        3:
	            IF #bCanActive THEN
	                IF NOT (#arrRecord[0] = 's' AND
	                    #arrRecord[12] = 'A' AND
	                    #arrRecord[13] = 'N' AND
	                    #arrRecord[23] = 'a' AND
	                    #arrRecord[24] = 'l' AND
	                    #arrRecord[25] = 'l' AND
	                    #arrRecord[26] = ' ' AND
	                    #arrRecord[27] = '1') THEN

	                    #nTempErrorCode := 16#0000_0016; (*Error: Invalid device answer*)
	                END_IF;
	            ELSE
	                IF NOT (#arrRecord[0] = 's' AND
	                    #arrRecord[1] = 'A' AND
	                    #arrRecord[2] = 'N' AND
	                    #arrRecord[12] = 'a' AND
	                    #arrRecord[13] = 'l' AND
	                    #arrRecord[14] = 'l' AND
	                    #arrRecord[15] = ' ' AND
	                    #arrRecord[16] = '1') THEN

	                    #nTempErrorCode := 16#0000_0016; (*Error: Invalid device answer*)
	                END_IF;
	            END_IF;

	            IF #nTempErrorCode = 0 THEN
	                #iCommandIndex := 11; (*Logout*)
	                #iStep := 4;         (*Create command*)
	            END_IF;

	            (*Check "Communication Test" response*)
	        4:
	            IF #bCanActive THEN
	                IF #arrRecord[0] = 's' AND
	                    #arrRecord[12] = 'R' AND
	                    #arrRecord[13] = 'A' AND
	                    #arrRecord[14] = ' ' THEN

	                    #iStep := 8; (*Action performed*)
	                ELSE
	                    #nTempErrorCode := 16#0000_0016; (*Error: Invalid device answer*)
	                END_IF;
	            ELSE
	                IF #arrRecord[0] = 's' AND
	                    #arrRecord[1] = 'R' AND
	                    #arrRecord[2] = 'A' AND
	                    #arrRecord[3] = ' ' THEN

	                    #iStep := 8; (*Action performed*)
	                ELSE
	                    #nTempErrorCode := 16#0000_0016; (*Error: Invalid device answer*)
	                END_IF;
	            END_IF;

	            (*Check "Free command" response*)
	        5:
	            IF #fbCCom.ReqLength <= MAX_LEN(#Data.FreeCommand.sResult) THEN
	                Chars_TO_Strg(Chars := #arrRecord,
	                              pChars := 0,
	                              Cnt := INT_TO_UINT(#fbCCom.ReqLength),
	                              Strg => #Data.FreeCommand.sResult);
	                #iStep := 8; (*Action performed*)
	            ELSE
	                #nTempErrorCode := 16#0000_0021; (*Error: Free command result > Result string*)
	            END_IF;

	            (*Check "Login" response*)
	        10:
	            IF #bCanActive THEN
	                IF NOT (#arrRecord[0] = 's' AND
	                    #arrRecord[12] = 'A' AND
	                    #arrRecord[13] = 'N' AND
	                    #arrRecord[24] = 'M' AND
	                    #arrRecord[25] = 'o' AND
	                    #arrRecord[26] = 'd' AND
	                    #arrRecord[27] = 'e' AND
	                    #arrRecord[28] = ' ' AND
	                    #arrRecord[29] = '1') THEN

	                    #nTempErrorCode := 16#0000_0016; (*Error: Invalid device answer*)
	                END_IF;
	            ELSE
	                IF NOT (#arrRecord[0] = 's' AND
	                    #arrRecord[1] = 'A' AND
	                    #arrRecord[2] = 'N' AND
	                    #arrRecord[13] = 'M' AND
	                    #arrRecord[14] = 'o' AND
	                    #arrRecord[15] = 'd' AND
	                    #arrRecord[16] = 'e' AND
	                    #arrRecord[17] = ' ' AND
	                    #arrRecord[18] = '1') THEN

	                    #nTempErrorCode := 16#0000_0016; (*Error: Invalid device answer*)
	                END_IF;
	            END_IF;

	            IF #nTempErrorCode = 0 THEN
	                IF #arrSelection[2] THEN
	                    #iCommandIndex := 2; (*Matchcode*)
	                    #iStep := 4;         (*Create command*)
	                ELSIF #arrSelection[3] THEN
	                    #iCommandIndex := 3; (*Save permanent*)
	                    #iStep := 4;         (*Create command*)
	                END_IF;
	                #bDeviceState := true; (*Edit-Mode active*)
	            END_IF;

	            (*Check "Logout" response*)
	        11:
	            IF #bCanActive THEN
	                IF #arrRecord[0] = 's' AND
	                    #arrRecord[12] = 'A' AND
	                    #arrRecord[13] = 'N' AND
	                    #arrRecord[14] = ' ' AND
	                    #arrRecord[15] = 'R' AND
	                    #arrRecord[16] = 'u' AND
	                    #arrRecord[17] = 'n' AND
	                    #arrRecord[18] = ' ' AND
	                    #arrRecord[19] = '1' THEN

	                    #bDeviceState := false; (*Run-Mode active*)
	                    #iStep := 8; (*Action performed*)
	                ELSE
	                    #nTempErrorCode := 16#0000_0016; (*Error: Invalid device answer*)
	                END_IF;
	            ELSE
	                IF #arrRecord[0] = 's' AND
	                    #arrRecord[1] = 'A' AND
	                    #arrRecord[2] = 'N' AND
	                    #arrRecord[3] = ' ' AND
	                    #arrRecord[4] = 'R' AND
	                    #arrRecord[5] = 'u' AND
	                    #arrRecord[6] = 'n' AND
	                    #arrRecord[7] = ' ' AND
	                    #arrRecord[8] = '1' THEN

	                    #bDeviceState := false; (*Run-Mode active*)
	                    #iStep := 8; (*Action performed*)
	                ELSE
	                    #nTempErrorCode := 16#0000_0016; (*Error: Invalid device answer*)
	                END_IF;
	            END_IF;
	    END_CASE;
	END_IF;


	(*================================ ACTION PERFORMED (STEP 8) ===============================*)
	IF #iStep = 8 THEN
	    IF #bEnforceLogout THEN
	        #nTempErrorCode := #nLogoutErrorCode;
	    ELSE
	        #ReqDone := true;
	        #ReqBusy := false;
	        #bReqBusyMem := false;
	        #iStep := 0;
	    END_IF;
	END_IF;


	(*====================================== COMMUNICATION =====================================*)
	#fbCCom(HWInputIdent := #HWInputIdent,
	        HWInputLength := #HWInputLength,
	        HWOutputIdent := #HWOutputIdent,
	        HWOutputLength := #HWOutputLength,
	        TOut := #TOut + T#1s,
	        CommandLength := #iCommandLength,
	        arrCommand := #arrCommand,
	        arrRecord := #arrRecord);

	(*Reset the request flag every cycle*)
	#fbCCom.Req := false;

	(*Read result error*)
	IF #fbCCom.RdLength < 0 AND #fbCCom.RdDone THEN
	    #Data.ReadingResult.iLength := -1; (*Error: Reading result longer than record array*)
	    FOR #iTemp1 := 1 TO UINT_TO_INT(#iReadingResultSize) DO
	        #Data.ReadingResult.arrResult[#iTemp1] := 16#00;
	    END_FOR;

	(*Handling of the reading result*)
	ELSIF #fbCCom.RdDone THEN
	    IF #fbCCom.RdLength > #iReadingResultSize THEN
	        #Data.ReadingResult.iLength := -1; (*Error: Reading result longer than reading result array*)
	        FOR #iTemp1 := 1 TO UINT_TO_INT(#iReadingResultSize) DO
	            #Data.ReadingResult.arrResult[#iTemp1] := 16#00;
	        END_FOR;
	    ELSE
	        MOVE_BLK(IN := #arrRecord[0],
	                 COUNT := INT_TO_UINT(#fbCCom.RdLength),
	                 OUT => #Data.ReadingResult.arrResult[1]);
	        IF (#Data.ReadingResult.iCounter >= 255) THEN
	            #Data.ReadingResult.iCounter := 0;
	        ELSE
	            #Data.ReadingResult.iCounter := #Data.ReadingResult.iCounter + 1;
	        END_IF;
	        #Data.ReadingResult.iLength := #fbCCom.RdLength;
	        #RdDone := true;
	    END_IF;
	END_IF;
END_FUNCTION_BLOCK

TYPE "UDT_Message"
TITLE = UDT_Message
VERSION : 0.1
//User-defined structure of the message characters array.
   STRUCT
      Character : Array[0..499] of Char;   // Message character
   END_STRUCT;

END_TYPE

TYPE "UDT_HMMessageHeader"
TITLE = UDT_H&MMessage
VERSION : 0.1
//User-defined structure of H&M message data.
   STRUCT
      STX { ExternalAccessible := 'False'; ExternalVisible := 'False'; ExternalWritable := 'False'} : Char;
      PLCID : String[4];   // Integer that globally identifies the connection
      SequenceNumber : String[8];   // Padded with leading zeros (8 characters total)
      MessageHeader : String[15];   // Message type defined by header
   END_STRUCT;

END_TYPE

FUNCTION "FC_BitAllocation" : Void
{ S7_Optimized_Access := 'TRUE' }
VERSION : 0.1
   VAR_INPUT
      ix_Bit0 : Bool;
      ix_Bit1 : Bool;
      ix_Bit2 : Bool;
      ix_Bit3 : Bool;
      ix_Bit4 : Bool;
      ix_Bit5 : Bool;
      ix_Bit6 : Bool;
      ix_Bit7 : Bool;
      ix_Bit8 : Bool;
      ix_Bit9 : Bool;
      ix_Bit10 : Bool;
      ix_Bit11 : Bool;
      ix_Bit12 : Bool;
      ix_Bit13 : Bool;
      ix_Bit14 : Bool;
      ix_Bit15 : Bool;
      ix_Bit16 : Bool;
      ix_Bit17 : Bool;
      ix_Bit18 : Bool;
      ix_Bit19 : Bool;
      ix_Bit20 : Bool;
      ix_Bit21 : Bool;
      ix_Bit22 : Bool;
      ix_Bit23 : Bool;
      ix_Bit24 : Bool;
      ix_Bit25 : Bool;
      ix_Bit26 : Bool;
      ix_Bit27 : Bool;
      ix_Bit28 : Bool;
      ix_Bit29 : Bool;
      ix_Bit30 : Bool;
      ix_Bit31 : Bool;
   END_VAR

   VAR_OUTPUT
      qdw_Dword : DWord;
   END_VAR


BEGIN
	#qdw_Dword.%X0 := #ix_Bit0;
	#qdw_Dword.%X1 := #ix_Bit1;
	#qdw_Dword.%X2 := #ix_Bit2;
	#qdw_Dword.%X3 := #ix_Bit3;
	#qdw_Dword.%X4 := #ix_Bit4;
	#qdw_Dword.%X5 := #ix_Bit5;
	#qdw_Dword.%X6 := #ix_Bit6;
	#qdw_Dword.%X7 := #ix_Bit7;
	#qdw_Dword.%X8 := #ix_Bit8;
	#qdw_Dword.%X9 := #ix_Bit9;
	#qdw_Dword.%X10 := #ix_Bit10;
	#qdw_Dword.%X11 := #ix_Bit11;
	#qdw_Dword.%X12 := #ix_Bit12;
	#qdw_Dword.%X13 := #ix_Bit13;
	#qdw_Dword.%X14 := #ix_Bit14;
	#qdw_Dword.%X15 := #ix_Bit15;
	#qdw_Dword.%X16 := #ix_Bit16;
	#qdw_Dword.%X17 := #ix_Bit17;
	#qdw_Dword.%X18 := #ix_Bit18;
	#qdw_Dword.%X19 := #ix_Bit19;
	#qdw_Dword.%X20 := #ix_Bit20;
	#qdw_Dword.%X21 := #ix_Bit21;
	#qdw_Dword.%X22 := #ix_Bit22;
	#qdw_Dword.%X23 := #ix_Bit23;
	#qdw_Dword.%X24 := #ix_Bit24;
	#qdw_Dword.%X25 := #ix_Bit25;
	#qdw_Dword.%X26 := #ix_Bit26;
	#qdw_Dword.%X27 := #ix_Bit27;
	#qdw_Dword.%X28 := #ix_Bit28;
	#qdw_Dword.%X29 := #ix_Bit29;
	#qdw_Dword.%X30 := #ix_Bit30;
	#qdw_Dword.%X31 := #ix_Bit31;

END_FUNCTION

TYPE "UDT_DataLogic_OUT"
VERSION : 0.1
   STRUCT
      "Unused_0.0" : Bool;   // Unused
      "Unused_0.1" : Bool;   // Unused
      "Unused_0.2" : Bool;   // Unused
      "Unused_0.3" : Bool;   // Unused
      "Unused_0.4" : Bool;   // Unused
      "Unused_0.5" : Bool;   // Unused
      "Unused_0.6" : Bool;   // Unused
      BladeTrigger : Bool;   // Camera input for trigger
      Unused_1 : Byte;   // Unused
      UnusedBytes : Array[0..14] of Byte;   // Unused
   END_STRUCT;

END_TYPE

TYPE "UDT_StatisticsTC36"
VERSION : 0.1
//Two direction, motor, Tracking, popup, pos. Switch
   STRUCT
      RightAngledTransfer : "UDT_RATStatistics";   // Right angled transfer Statistics
      MCO_M01 : "UDT_VfdStatistics";   // MCO Statistics
   END_STRUCT;

END_TYPE

FUNCTION "FC_WriteGIN" : Void
{ S7_Optimized_Access := 'TRUE' }
VERSION : 0.1
// ATTRIBUTES
// AUTO_NUMBER = True
// BLOCK_NUMBER = 31
// END_ATTRIBUTES
   VAR_INPUT
      ii_GIN : Int;   //    GIN number
      ii_PositionToWrite : Int;   //    Position in tracking array where to start writing GIN
      ii_NumberOfPositions : Int;   //    Number of positions to be written
      ix_Direction : Bool;   //    TRUE when positions in positive direction have to be written
   END_VAR

   VAR_IN_OUT
      iqa_TrackingData : Array[*] of Int;   //    Tracking data
   END_VAR

   VAR_TEMP
      ti_LCWritePosition : Int;   //    Loop counter
   END_VAR


BEGIN
	(*
	----------------------------------------------------------------------------------------

	Version history:
	Date        | Version   | Author        | Remark
	----------------------------------------------------------------------------------------
	27/02/2020  | 3.1       | L.Klar        | first release MHSE TIA 15.1
	21/02/2023  | 4.0       | F.Baten       | 4.0 Release TIA 17.5
	*)

	REGION 1 – GIN write

	    // Depending on the direction, a GIN is written into a specific number of tracking array positions.
	    #ti_LCWritePosition := 0;

	    IF #ix_Direction
	    THEN
	        FOR #ti_LCWritePosition := #ii_PositionToWrite TO #ii_PositionToWrite + #ii_NumberOfPositions - 1 BY 1 DO
	            #iqa_TrackingData[#ti_LCWritePosition] := #ii_GIN;
	        END_FOR;
	    ELSE
	        FOR #ti_LCWritePosition := #ii_PositionToWrite TO #ii_PositionToWrite - #ii_NumberOfPositions + 1 BY -1 DO
	            #iqa_TrackingData[#ti_LCWritePosition] := #ii_GIN;
	        END_FOR;
	    END_IF;

	END_REGION
END_FUNCTION

TYPE "UDT_VfdNordPO"
TITLE = UDT_VfdNordPO
VERSION : 0.1
//User-defined structure of VFD Nord output telegram.
   STRUCT
      STW : Struct   // Control Word
         "StartFunction408.11" { ExternalAccessible := 'False'; ExternalVisible := 'False'; ExternalWritable := 'False'} : Bool;   // 1 = Bus bit 8 of control word is set. P480
         "StartFunction408.12" { ExternalAccessible := 'False'; ExternalVisible := 'False'; ExternalWritable := 'False'} : Bool;   // 1 = Bus bit 8 of control word is set. P480
         ControlDataValid { ExternalAccessible := 'False'; ExternalVisible := 'False'; ExternalWritable := 'False'} : Bool;   // 1 = The bus master trasnfers valid process data. 0 = The transmitted process data are invalid
         RotationRightOn { ExternalAccessible := 'False'; ExternalVisible := 'False'; ExternalWritable := 'False'} : Bool;   // 1 = Switch on rotation right
         RotationLeftOn { ExternalAccessible := 'False'; ExternalVisible := 'False'; ExternalWritable := 'False'} : Bool;   // 1 = Switch on rotation left
         Reserved { ExternalAccessible := 'False'; ExternalVisible := 'False'; ExternalWritable := 'False'} : Bool;   // Reserved from NORD
         ParameterSetBit0 { ExternalAccessible := 'False'; ExternalVisible := 'False'; ExternalWritable := 'False'} : Bool;   // Activates parameter set
         ParameterSetBit1 { ExternalAccessible := 'False'; ExternalVisible := 'False'; ExternalWritable := 'False'} : Bool;   // Activates parameter set
         ReadyForOperation { ExternalAccessible := 'False'; ExternalVisible := 'False'; ExternalWritable := 'False'} : Bool;   // 1 = Set the frequency inverter to standby. 0=Reverse with brake ramp
         DisableVoltage { ExternalAccessible := 'False'; ExternalVisible := 'False'; ExternalWritable := 'False'} : Bool;   // 0 = Switch off the frequency inverter output voltage. 1 = Cancel "Disable voltage"
         EmergencyStop { ExternalAccessible := 'False'; ExternalVisible := 'False'; ExternalWritable := 'False'} : Bool;   // 0 = Emergency stop with programmed estop time. Not Fail Safe Estop. 1 = Cancel condition "Emergency stop"
         EnableOperation { ExternalAccessible := 'False'; ExternalVisible := 'False'; ExternalWritable := 'False'} : Bool;   // 1 = Enable output voltage acceleration to setpoint. 0 = Block voltage, switch off output voltage
         EnablePulsles { ExternalAccessible := 'False'; ExternalVisible := 'False'; ExternalWritable := 'False'} : Bool;   // 1 = Enable acceleration encoder. 0 = Acceleraton encoder is set to zero
         EnableRamp { ExternalAccessible := 'False'; ExternalVisible := 'False'; ExternalWritable := 'False'} : Bool;   // 1 = Enable setpoint on acceleration encoder. 0 = Freeze the setpoint provided by the acceleration encoder
         EnableSetpoint { ExternalAccessible := 'False'; ExternalVisible := 'False'; ExternalWritable := 'False'} : Bool;   // 1 = Activate the selected setpoint on the acceleration encoder. 0= Set the selected setpoint on the acceleration encoder to 0
         Acknowledge { ExternalAccessible := 'False'; ExternalVisible := 'False'; ExternalWritable := 'False'} : Bool;   // 0-->1 = Inactive errors are acknowledged
      END_STRUCT;
      FrequencySetPoint : Int;   // Frequency HZ SetPoint to VFD 100%=4000HEX /16384 DEC . 0% = 0000HEX / 0 DEC Normalization with P105
      RampTimeSetPoint : Int;   // Ramp time to VFD [Range 0..200%][100% = 4000HEX /16384DEC = 10sec]
   END_STRUCT;

END_TYPE

TYPE "UDT_AixPlcFullOut"
VERSION : 0.1
   STRUCT
      ConveyStopControl { ExternalVisible := 'False'} : Word;   // Writing '1' causes the Stop group to go into STOP state . Transition 0 - 2 is needed to clear the Stop
      LeftMotorAsDIO { ExternalVisible := 'False'} : Struct   // Use the Left M8 motor port as digital IO
         Bit08 { ExternalAccessible := 'False'; ExternalVisible := 'False'; ExternalWritable := 'False'} : Bool;   // Reserved
         Bit09 { ExternalAccessible := 'False'; ExternalVisible := 'False'; ExternalWritable := 'False'} : Bool;   // Reserved
         Bit10 { ExternalAccessible := 'False'; ExternalVisible := 'False'; ExternalWritable := 'False'} : Bool;   // Reserved
         Bit11 { ExternalAccessible := 'False'; ExternalVisible := 'False'; ExternalWritable := 'False'} : Bool;   // Reserved
         Bit12 { ExternalAccessible := 'False'; ExternalVisible := 'False'; ExternalWritable := 'False'} : Bool;   // Reserved
         Bit13 { ExternalAccessible := 'False'; ExternalVisible := 'False'; ExternalWritable := 'False'} : Bool;   // Reserved
         Bit14 { ExternalAccessible := 'False'; ExternalVisible := 'False'; ExternalWritable := 'False'} : Bool;   // Reserved
         EnableDIO { ExternalAccessible := 'False'; ExternalVisible := 'False'; ExternalWritable := 'False'} : Bool;   // Set bit to enable Left motor M8 port Digital IO mode
         Bit00 { ExternalAccessible := 'False'; ExternalVisible := 'False'; ExternalWritable := 'False'} : Bool;   // Reserved
         EnergizeM8Pin4 { ExternalAccessible := 'False'; ExternalVisible := 'False'; ExternalWritable := 'False'} : Bool;   // Energize motor port M8 PIN 4
         EnergizeM8Pin3 { ExternalAccessible := 'False'; ExternalVisible := 'False'; ExternalWritable := 'False'} : Bool;   // Energize motor port M8 PIN 3
         Bit03 { ExternalAccessible := 'False'; ExternalVisible := 'False'; ExternalWritable := 'False'} : Bool;   // Reserved
         Bit04 { ExternalAccessible := 'False'; ExternalVisible := 'False'; ExternalWritable := 'False'} : Bool;   // Reserved
         Bit05 { ExternalAccessible := 'False'; ExternalVisible := 'False'; ExternalWritable := 'False'} : Bool;   // Reserved
         Bit06 { ExternalAccessible := 'False'; ExternalVisible := 'False'; ExternalWritable := 'False'} : Bool;   // Reserved
         Bit07 { ExternalAccessible := 'False'; ExternalVisible := 'False'; ExternalWritable := 'False'} : Bool;   // Reserved
      END_STRUCT;
      RightMotorAsDIO { ExternalVisible := 'False'} : Struct   // Use the Right M8 motor port as digital IO
         Bit08 { ExternalAccessible := 'False'; ExternalVisible := 'False'; ExternalWritable := 'False'} : Bool;   // Reserved
         Bit09 { ExternalAccessible := 'False'; ExternalVisible := 'False'; ExternalWritable := 'False'} : Bool;   // Reserved
         Bit10 { ExternalAccessible := 'False'; ExternalVisible := 'False'; ExternalWritable := 'False'} : Bool;   // Reserved
         Bit11 { ExternalAccessible := 'False'; ExternalVisible := 'False'; ExternalWritable := 'False'} : Bool;   // Reserved
         Bit12 { ExternalAccessible := 'False'; ExternalVisible := 'False'; ExternalWritable := 'False'} : Bool;   // Reserved
         Bit13 { ExternalAccessible := 'False'; ExternalVisible := 'False'; ExternalWritable := 'False'} : Bool;   // Reserved
         Bit14 { ExternalAccessible := 'False'; ExternalVisible := 'False'; ExternalWritable := 'False'} : Bool;   // Reserved
         EnableDIO { ExternalAccessible := 'False'; ExternalVisible := 'False'; ExternalWritable := 'False'} : Bool;   // Set bit to enable Left motor M8 port Digital IO mode
         EnergizeM8Pin2 { ExternalAccessible := 'False'; ExternalVisible := 'False'; ExternalWritable := 'False'} : Bool;   // Energize motor port M8 PIN 2
         Bit01 { ExternalAccessible := 'False'; ExternalVisible := 'False'; ExternalWritable := 'False'} : Bool;   // Reserved
         EnergizeM8Pin3 { ExternalAccessible := 'False'; ExternalVisible := 'False'; ExternalWritable := 'False'} : Bool;   // Energize motor port M8 PIN 3
         Bit03 { ExternalAccessible := 'False'; ExternalVisible := 'False'; ExternalWritable := 'False'} : Bool;   // Reserved
         Bit04 { ExternalAccessible := 'False'; ExternalVisible := 'False'; ExternalWritable := 'False'} : Bool;   // Reserved
         Bit05 { ExternalAccessible := 'False'; ExternalVisible := 'False'; ExternalWritable := 'False'} : Bool;   // Reserved
         Bit06 { ExternalAccessible := 'False'; ExternalVisible := 'False'; ExternalWritable := 'False'} : Bool;   // Reserved
         Bit07 { ExternalAccessible := 'False'; ExternalVisible := 'False'; ExternalWritable := 'False'} : Bool;   // Reserved
      END_STRUCT;
      SensorPortsDO { ExternalVisible := 'False'} : Struct   // The Sensor ports PIN2 as digital outputs
         Bit08 { ExternalAccessible := 'False'; ExternalVisible := 'False'; ExternalWritable := 'False'} : Bool;   // Reserved
         Bit09 { ExternalAccessible := 'False'; ExternalVisible := 'False'; ExternalWritable := 'False'} : Bool;   // Reserved
         Bit10 { ExternalAccessible := 'False'; ExternalVisible := 'False'; ExternalWritable := 'False'} : Bool;   // Reserved
         Bit11 { ExternalAccessible := 'False'; ExternalVisible := 'False'; ExternalWritable := 'False'} : Bool;   // Reserved
         Bit12 { ExternalAccessible := 'False'; ExternalVisible := 'False'; ExternalWritable := 'False'} : Bool;   // Reserved
         Bit13 { ExternalAccessible := 'False'; ExternalVisible := 'False'; ExternalWritable := 'False'} : Bool;   // Reserved
         Bit14 { ExternalAccessible := 'False'; ExternalVisible := 'False'; ExternalWritable := 'False'} : Bool;   // Reserved
         Bit15 { ExternalAccessible := 'False'; ExternalVisible := 'False'; ExternalWritable := 'False'} : Bool;   // Reserved
         EnergizeLeftPortPin2 { ExternalAccessible := 'False'; ExternalVisible := 'False'; ExternalWritable := 'False'} : Bool;   // Set to turn on Left Port Pin2
         EnergizeRightPortPin2 { ExternalAccessible := 'False'; ExternalVisible := 'False'; ExternalWritable := 'False'} : Bool;   // Set to turn on Right Port Pin2
         Bit02 { ExternalAccessible := 'False'; ExternalVisible := 'False'; ExternalWritable := 'False'} : Bool;   // Reserved
         Bit03 { ExternalAccessible := 'False'; ExternalVisible := 'False'; ExternalWritable := 'False'} : Bool;   // Reserved
         Bit04 { ExternalAccessible := 'False'; ExternalVisible := 'False'; ExternalWritable := 'False'} : Bool;   // Reserved
         EnableLeftPortPin2 { ExternalAccessible := 'False'; ExternalVisible := 'False'; ExternalWritable := 'False'} : Bool;   // Set to enable, reset for Pin2  to be input
         EnableRightPortPin2 { ExternalAccessible := 'False'; ExternalVisible := 'False'; ExternalWritable := 'False'} : Bool;   // Set to enable, reset for Pin2  to be input
         Bit07 { ExternalAccessible := 'False'; ExternalVisible := 'False'; ExternalWritable := 'False'} : Bool;   // Reserved
      END_STRUCT;
      LeftMotorControl { ExternalVisible := 'False'} : Struct   // Run/Stop and Direction control of the Left motor
         MotorDirection { ExternalAccessible := 'False'; ExternalVisible := 'False'; ExternalWritable := 'False'} : Bool;   // 0 = Configured direction /1 = opposite to configured direction
         Bit09 { ExternalAccessible := 'False'; ExternalVisible := 'False'; ExternalWritable := 'False'} : Bool;   // Reserved
         Bit10 { ExternalAccessible := 'False'; ExternalVisible := 'False'; ExternalWritable := 'False'} : Bool;   // Reserved
         Bit11 { ExternalAccessible := 'False'; ExternalVisible := 'False'; ExternalWritable := 'False'} : Bool;   // Reserved
         Bit12 { ExternalAccessible := 'False'; ExternalVisible := 'False'; ExternalWritable := 'False'} : Bool;   // Reserved
         Bit13 { ExternalAccessible := 'False'; ExternalVisible := 'False'; ExternalWritable := 'False'} : Bool;   // Reserved
         Bit14 { ExternalAccessible := 'False'; ExternalVisible := 'False'; ExternalWritable := 'False'} : Bool;   // Reserved
         Bit15 { ExternalAccessible := 'False'; ExternalVisible := 'False'; ExternalWritable := 'False'} : Bool;   // Reserved
         Run { ExternalAccessible := 'False'; ExternalVisible := 'False'; ExternalWritable := 'False'} : Bool;   // Run = 1 / Stop = 0
         Bit01 { ExternalAccessible := 'False'; ExternalVisible := 'False'; ExternalWritable := 'False'} : Bool;   // Reserved
         Bit02 { ExternalAccessible := 'False'; ExternalVisible := 'False'; ExternalWritable := 'False'} : Bool;   // Reserved
         Bit03 { ExternalAccessible := 'False'; ExternalVisible := 'False'; ExternalWritable := 'False'} : Bool;   // Reserved
         Bit04 { ExternalAccessible := 'False'; ExternalVisible := 'False'; ExternalWritable := 'False'} : Bool;   // Reserved
         Bit05 { ExternalAccessible := 'False'; ExternalVisible := 'False'; ExternalWritable := 'False'} : Bool;   // Reserved
         Bit06 { ExternalAccessible := 'False'; ExternalVisible := 'False'; ExternalWritable := 'False'} : Bool;   // Reserved
         Bit07 { ExternalAccessible := 'False'; ExternalVisible := 'False'; ExternalWritable := 'False'} : Bool;   // Reserved
      END_STRUCT;
      LeftSetMotorBrakeMode { ExternalVisible := 'False'} : Word;   // Set Left motor Brake Mode.0 = ignore 1 = "Normal" / 2 = "Free" / 3 ="Servo brake"
      LeftSetMotorSlaveMode { ExternalVisible := 'False'} : Word;   // 0 = ignore  1=Off, Left Independant  2=On, Left Mirror Right   3=On, Left Opposite Right direction
      RightMotorControl { ExternalVisible := 'False'} : Struct   // Run/Stop and Direction control of the Right motor
         MotorDirection { ExternalAccessible := 'False'; ExternalVisible := 'False'; ExternalWritable := 'False'} : Bool;   // 0 = Configured direction /1 = opposite to configured direction
         Bit09 { ExternalAccessible := 'False'; ExternalVisible := 'False'; ExternalWritable := 'False'} : Bool;   // Reserved
         Bit10 { ExternalAccessible := 'False'; ExternalVisible := 'False'; ExternalWritable := 'False'} : Bool;   // Reserved
         Bit11 { ExternalAccessible := 'False'; ExternalVisible := 'False'; ExternalWritable := 'False'} : Bool;   // Reserved
         Bit12 { ExternalAccessible := 'False'; ExternalVisible := 'False'; ExternalWritable := 'False'} : Bool;   // Reserved
         Bit13 { ExternalAccessible := 'False'; ExternalVisible := 'False'; ExternalWritable := 'False'} : Bool;   // Reserved
         Bit14 { ExternalAccessible := 'False'; ExternalVisible := 'False'; ExternalWritable := 'False'} : Bool;   // Reserved
         Bit15 { ExternalAccessible := 'False'; ExternalVisible := 'False'; ExternalWritable := 'False'} : Bool;   // Reserved
         Run { ExternalAccessible := 'False'; ExternalVisible := 'False'; ExternalWritable := 'False'} : Bool;   // Run = 1 / Stop = 0
         Bit01 { ExternalAccessible := 'False'; ExternalVisible := 'False'; ExternalWritable := 'False'} : Bool;   // Reserved
         Bit02 { ExternalAccessible := 'False'; ExternalVisible := 'False'; ExternalWritable := 'False'} : Bool;   // Reserved
         Bit03 { ExternalAccessible := 'False'; ExternalVisible := 'False'; ExternalWritable := 'False'} : Bool;   // Reserved
         Bit04 { ExternalAccessible := 'False'; ExternalVisible := 'False'; ExternalWritable := 'False'} : Bool;   // Reserved
         Bit05 { ExternalAccessible := 'False'; ExternalVisible := 'False'; ExternalWritable := 'False'} : Bool;   // Reserved
         Bit06 { ExternalAccessible := 'False'; ExternalVisible := 'False'; ExternalWritable := 'False'} : Bool;   // Reserved
         Bit07 { ExternalAccessible := 'False'; ExternalVisible := 'False'; ExternalWritable := 'False'} : Bool;   // Reserved
      END_STRUCT;
      RightSetMotorBrakeMode { ExternalVisible := 'False'} : Word;   // Set Right motor Brake Mode.0 = ignore 1 = "Normal" / 2 = "Free" / 3 ="Servo brake"
      RightSetMotorSlaveMode { ExternalVisible := 'False'} : Word;   // 0 = ignore 1=Off, Right Independant  2=On, Right Mirror Right   3=On, Right Opposite Right direction
      LeftSetMotorSpeed { ExternalVisible := 'False'} : Int;   // Set reference speed for Left motor in mm/s (or 1/10 of an RPM for PGD)
      RightSetMotorSpeed { ExternalVisible := 'False'} : Int;   // Set reference speed for Right motor mm/s  (or 1/10 of an RPM for PGD)
      LeftSetMotorAccel { ExternalVisible := 'False'} : Int;   // Set acceleration distance in mm for Left motor (or pulses for PGD)
      LeftSetMotorDeccel { ExternalVisible := 'False'} : Int;   // Set deceleration distance in mm for Left motor (or pulses for PGD)
      RightSetMotorAccel { ExternalVisible := 'False'} : Int;   // Set acceleration distance in mm for Right motor (or pulses for PGD)
      RightSetMotorDeccel { ExternalVisible := 'False'} : Int;   // Set deceleration distance in mm for Right motor (or pulses for PGD)
      ClearMotorError { ExternalVisible := 'False'} : Word;   // Write '1' to clear motor error, wait 500 msec, then write '0' return to operation
      SendStatusToDownstream { ExternalVisible := 'False'} : Word;   // Write '4' or '5' to signal downstream ConveyLinx module in ZPA mode to wake up
      SendStatusToUpstream { ExternalVisible := 'False'} : Word;   // Write '5' to signal upstream ConveyLinx module in ZPA mode to accumulate, write '1' to signal OK to receive
      SensorPolarity { ExternalVisible := 'False'} : Struct   // Set logic polarity for Sensor Port's PIN2 and PIN4
         Bit08 { ExternalAccessible := 'False'; ExternalVisible := 'False'; ExternalWritable := 'False'} : Bool;   // Reserved
         Bit09 { ExternalAccessible := 'False'; ExternalVisible := 'False'; ExternalWritable := 'False'} : Bool;   // Reserved
         Bit10 { ExternalAccessible := 'False'; ExternalVisible := 'False'; ExternalWritable := 'False'} : Bool;   // Reserved
         Bit11 { ExternalAccessible := 'False'; ExternalVisible := 'False'; ExternalWritable := 'False'} : Bool;   // Reserved
         Bit12 { ExternalAccessible := 'False'; ExternalVisible := 'False'; ExternalWritable := 'False'} : Bool;   // Reserved
         Bit13 { ExternalAccessible := 'False'; ExternalVisible := 'False'; ExternalWritable := 'False'} : Bool;   // Reserved
         Bit14 { ExternalAccessible := 'False'; ExternalVisible := 'False'; ExternalWritable := 'False'} : Bool;   // Reserved
         Bit15 { ExternalAccessible := 'False'; ExternalVisible := 'False'; ExternalWritable := 'False'} : Bool;   // Reserved
         Left_Pin2 { ExternalAccessible := 'False'; ExternalVisible := 'False'; ExternalWritable := 'False'} : Bool;   // Set to invert, reset for normal
         Bit01 { ExternalAccessible := 'False'; ExternalVisible := 'False'; ExternalWritable := 'False'} : Bool;   // Reserved
         Right_Pin2 { ExternalAccessible := 'False'; ExternalVisible := 'False'; ExternalWritable := 'False'} : Bool;   // Set to invert, reset for normal
         Bit03 { ExternalAccessible := 'False'; ExternalVisible := 'False'; ExternalWritable := 'False'} : Bool;   // Reserved
         Left_Pin4 { ExternalAccessible := 'False'; ExternalVisible := 'False'; ExternalWritable := 'False'} : Bool;   // Set to invert, reset for normal
         Bit05 { ExternalAccessible := 'False'; ExternalVisible := 'False'; ExternalWritable := 'False'} : Bool;   // Reserved
         Right_Pin4 { ExternalAccessible := 'False'; ExternalVisible := 'False'; ExternalWritable := 'False'} : Bool;   // Set to invert, reset for normal
         Bit07 { ExternalAccessible := 'False'; ExternalVisible := 'False'; ExternalWritable := 'False'} : Bool;   // Reserved
      END_STRUCT;
      TrackingToDownstream { ExternalVisible := 'False'} : DWord;   // Write Tracking data to be captured by downstream ZPA mode ConveyLinx
      Index22 { ExternalVisible := 'False'} : Word;   // Reserved
      ServoControlDistanceLeft { ExternalVisible := 'False'} : Int;   // Position from 0 in mm for Left motor to move on next command
      ServoControlCommandLeft { ExternalVisible := 'False'} : Word;   // Left motor servo command
      ServoControlDistanceRight { ExternalVisible := 'False'} : Int;   // New position from 0 in mm for Right motor to move on next command
      ServoControlCommandRight { ExternalVisible := 'False'} : Word;   // Right motor servo command
      Future { ExternalVisible := 'False'} : Array[27..31] of Int;   // Reserved
   END_STRUCT;

END_TYPE

